// TwinCAT 3 PLC project NUCOIL
// libraries:
//   TcSUPS_CX51x0,newest,Evolution
//   YaskawaFunctions,newest,Evolution
//   Tc2_Drive, * (Beckhoff Automation GmbH)
//   Tc2_EtherCAT, * (Beckhoff Automation GmbH)
//   Tc2_IoFunctions, * (Beckhoff Automation GmbH)
//   Tc2_Math, * (Beckhoff Automation GmbH)
//   Tc2_MC2, * (Beckhoff Automation GmbH)
//   Tc2_MC2_Camming, * (Beckhoff Automation GmbH)
//   Tc2_NC, * (Beckhoff Automation GmbH)
//   Tc2_Standard, * (Beckhoff Automation GmbH)
//   Tc2_System, * (Beckhoff Automation GmbH)
//   Tc2_Utilities, * (Beckhoff Automation GmbH)
//   Tc3_Module, * (Beckhoff Automation GmbH)
// project tree:
//   Data types/ ST_AirTableBuf.TcDUT, ST_AlertLight.TcDUT, ST_AnaInput.TcDUT, ST_AxisPosBuf.TcDUT, ST_AxisTableBuf.TcDUT, ST_AxisTrqBuf.TcDUT, ST_AxisVelBuf.TcDUT, ST_BrakeParam.TcDUT, ST_Cam.TcDUT, ST_CamTable.TcDUT, ST_DigitInput.TcDUT, ST_DigitOutput.TcDUT, ST_DriveAlarmCode.TcDUT, ST_ExFSpdUpTableBuf.TcDUT, ST_FeederInProduce.TcDUT, ST_G5Config.TcDUT, ST_G5Status.TcDUT, ST_Homing.TcDUT, ST_InputState.TcDUT, ST_IOSwitch.TcDUT, ST_ManMove.TcDUT, ST_MasterAxisPos.TcDUT, ST_MasterAxisValue.TcDUT, ST_McFBInOutVar.TcDUT, ST_MCRelativeInput.TcDUT, ST_MCRelativeOutput.TcDUT, ST_McValue.TcDUT, ST_OIL.TcDUT, ST_OneLineAir.TcDUT, ST_OneLineTable.TcDUT, ST_ProAndManRelativeState.TcDUT, ST_Produce.TcDUT, ST_RingBuffer.TcDUT, ST_RingBufferIO.TcDUT, ST_RingBufferIOPart.TcDUT, ST_RingBufferPart.TcDUT, ST_SetPosByUI.TcDUT, ST_SlaveEcData.TcDUT, ST_SubProgramConfig.TcDUT, ST_SubProgramTable.TcDUT, ST_Touch.TcDUT, ST_TouchAdjustConfig.TcDUT, ST_TouchConfig.TcDUT, ST_TouchProbe.TcDUT, ST_TouchProbeHomeByUI.TcDUT, ST_TouchTableBuf.TcDUT
//   Global Variables/ ENUMSTATE.TcDUT, Global_Variables.TcGVL, MachineSubTypeEnum.TcDUT, MachineTypeEnum.TcDUT, MANMOVEENUM.TcDUT, MotorVenderEnum.TcDUT, Variable_Configuration.TcGVL
//   POUs/ AlertLight.TcPOU, AxisStatusDataStore.TcPOU, CoEConfig.TcPOU, CommunicationQualityCheck.TcPOU, EMGStop.TcPOU, EncoderClear.TcPOU, Error.TcPOU, HomeByTouchProbe.TcPOU, IOMapping.TcPOU, MAIN.TcPOU, ManMove.TcPOU, MCRelativeMove.TcPOU, MoveToColPos.TcPOU, Mpg.TcPOU, prAxis.TcPOU, Produce.TcPOU, SetCountPosToActPos.TcPOU, SetOverride.TcPOU, SetPosByUI.TcPOU, SubRunAlone.TcPOU, UPS.TcPOU
//   POUs/FB/ AlarmListClear.TcPOU, FB_CheckInfoData.TcPOU, FB_CloseAir.TcPOU, FB_CloseIO.TcPOU, FB_CloseOil.TcPOU, FB_EcAbnormal.TcPOU, FB_EncoderClear.TcPOU, FB_FNeedHoldPos.TcPOU, FB_GetExtPosition.TcPOU, FB_GetMachineInfo.TcPOU, FB_InAnotherTouch.TcPOU, FB_IsAdjustAxis.TcPOU, FB_IsAdjustTouch.TcPOU, FB_PosNear.TcPOU, FB_ToubleShootIsError.TcPOU, FB_TouchEnd.TcPOU, FB_TouchProbe.TcPOU, ManMovCal.TcPOU, MasterMove.TcPOU, MasterMove2.TcPOU, PPMCal.TcPOU, RelativeMOVE.TcPOU, RelativeMOVE2.TcPOU, SetMotionFuction.TcPOU, SetPositionTable.TcPOU
//   / Standard.TcTTO
// real-time tasks:
//   TASK Standard: cycle T#1ms, priority 25, ADS port 350
// motion (NC):
//   TASK NC-Task 1 SAF: cycle T#1ms, priority 4, ADS port 501
//   TASK NC-Task 1 SVB: cycle T#10ms, priority 8, ADS port 511
//   AXIS Axis1 Slide1 (id 2)
//     Dynamic: AccelerationMaximum=0, DecelerationMaximum=0, Acceleration=233017000, Deceleration=233017000, Jerk=124275000000
//     Velo: Maximum=6553600
//     PositionAreaControl: Enable=false
//     TargetPosControl: Enable=false
//     encoder EncType=1
//       EncPara: ScaleFactorNumerator=1
//     drive DrvType=5
//       DrvPara: DriveControlDWord=#x00000001
//         Analog: VeloReferenz=6553600, TorqueSetpointScale=10, SmoothingFilterOrder=0, SmoothingFilterTime=0
//         TimeComp: TaskDelayCycles=1
//     controller CtrType=1
//       CtrPara: PriorControlFactor=1
//         PosDiffControl: Enable=false
//         Observer: BandWidth=20
//   AXIS Axis2 Slide2 (id 3)
//     Dynamic: AccelerationMaximum=0, DecelerationMaximum=0, Acceleration=699050750.00009, Deceleration=699050750.00009, Jerk=1118479200001.57
//     Velo: Maximum=6553600
//     PositionAreaControl: Enable=false
//     TargetPosControl: Enable=false
//     encoder EncType=1
//       EncPara: ScaleFactorNumerator=1
//     drive DrvType=5
//       DrvPara: DriveControlDWord=#x00000001
//         Analog: VeloReferenz=6553600, TorqueSetpointScale=10, SmoothingFilterOrder=0, SmoothingFilterTime=0
//         TimeComp: TaskDelayCycles=1
//     controller CtrType=1
//       CtrPara: PriorControlFactor=1
//         PosDiffControl: Enable=false
//         Observer: BandWidth=20
//   AXIS Axis3 Slide3 (id 4)
//     Dynamic: AccelerationMaximum=0, DecelerationMaximum=0, Acceleration=3019980000, Deceleration=3019980000, Jerk=3025310000000
//     Velo: Maximum=6553600
//     PositionAreaControl: Enable=false
//     TargetPosControl: Enable=false
//     encoder EncType=1
//       EncPara: ScaleFactorNumerator=1
//     drive DrvType=5
//       DrvPara: DriveControlDWord=#x00000001
//         Analog: VeloReferenz=6553600, TorqueSetpointScale=10, SmoothingFilterOrder=0, SmoothingFilterTime=0
//         TimeComp: TaskDelayCycles=1
//     controller CtrType=1
//       CtrPara: PriorControlFactor=1
//         PosDiffControl: Enable=false
//         Observer: BandWidth=20
//   AXIS Axis4 Slide4 (id 5)
//     Dynamic: AccelerationMaximum=0, DecelerationMaximum=0, Acceleration=2206380000, Deceleration=2206380000, Jerk=11142200000000
//     Velo: Maximum=6553600
//     PositionAreaControl: Enable=false
//     TargetPosControl: Enable=false
//     encoder EncType=1
//       EncPara: ScaleFactorNumerator=1
//     drive DrvType=5
//       DrvPara: DriveControlDWord=#x00000001
//         Analog: VeloReferenz=6553600, TorqueSetpointScale=10, SmoothingFilterOrder=0, SmoothingFilterTime=0
//         TimeComp: TaskDelayCycles=1
//     controller CtrType=1
//       CtrPara: PriorControlFactor=1
//         PosDiffControl: Enable=false
//         Observer: BandWidth=20
//   AXIS Axis5 Slide5 (id 6)
//     Dynamic: AccelerationMaximum=0, DecelerationMaximum=0, Acceleration=441276000, Deceleration=441276000, Jerk=2971260000000
//     Velo: Maximum=6553600
//     PositionAreaControl: Enable=false
//     TargetPosControl: Enable=false
//     encoder EncType=1
//       EncPara: ScaleFactorNumerator=1
//     drive DrvType=5
//       DrvPara: DriveControlDWord=#x00000001
//         Analog: VeloReferenz=6553600, TorqueSetpointScale=10, SmoothingFilterOrder=0, SmoothingFilterTime=0
//         TimeComp: TaskDelayCycles=1
//     controller CtrType=1
//       CtrPara: PriorControlFactor=1
//         PosDiffControl: Enable=false
//         Observer: BandWidth=20
//   AXIS Axis6 Slide6 (id 7)
//     Dynamic: AccelerationMaximum=0, DecelerationMaximum=0, Acceleration=2206380000, Deceleration=2206380000, Jerk=11142200000000
//     Velo: Maximum=6553600
//     PositionAreaControl: Enable=false
//     TargetPosControl: Enable=false
//     encoder EncType=1
//       EncPara: ScaleFactorNumerator=1
//     drive DrvType=5
//       DrvPara: DriveControlDWord=#x00000001
//         Analog: VeloReferenz=6553600, TorqueSetpointScale=10, SmoothingFilterOrder=0, SmoothingFilterTime=0
//         TimeComp: TaskDelayCycles=1
//     controller CtrType=1
//       CtrPara: PriorControlFactor=1
//         PosDiffControl: Enable=false
//         Observer: BandWidth=20
//   AXIS Axis7 Slide7 (id 8)
//     Dynamic: AccelerationMaximum=0, DecelerationMaximum=0, Acceleration=2206376778.77214, Deceleration=2206376778.77214, Jerk=11142167465677.8
//     Velo: Maximum=6553600
//     PositionAreaControl: Enable=false
//     TargetPosControl: Enable=false
//     encoder EncType=1
//       EncPara: ScaleFactorNumerator=1
//     drive DrvType=5
//       DrvPara: DriveControlDWord=#x00000001
//         Analog: VeloReferenz=6553600, TorqueSetpointScale=10, SmoothingFilterOrder=0, SmoothingFilterTime=0
//         TimeComp: TaskDelayCycles=1
//     controller CtrType=1
//       CtrPara: PriorControlFactor=1
//         PosDiffControl: Enable=false
//         Observer: BandWidth=20
//   AXIS Axis8 Slide8 (id 9)
//     Dynamic: AccelerationMaximum=0, DecelerationMaximum=0, Acceleration=2206376778.77214, Deceleration=2206376778.77214, Jerk=11142167465677.8
//     Velo: Maximum=6553600
//     PositionAreaControl: Enable=false
//     TargetPosControl: Enable=false
//     encoder EncType=1
//       EncPara: ScaleFactorNumerator=1
//     drive DrvType=5
//       DrvPara: DriveControlDWord=#x00000001
//         Analog: VeloReferenz=6553600, TorqueSetpointScale=10, SmoothingFilterOrder=0, SmoothingFilterTime=0
//         TimeComp: TaskDelayCycles=1
//     controller CtrType=1
//       CtrPara: PriorControlFactor=1
//         PosDiffControl: Enable=false
//         Observer: BandWidth=20
//   AXIS Axis9 Wire (id 10)
//     Dynamic: AccelerationMaximum=0, DecelerationMaximum=0, Acceleration=2206376778.77214, Deceleration=2206376778.77214, Jerk=11142167465677.8
//     Velo: Maximum=6553600
//     PositionAreaControl: Enable=false
//     TargetPosControl: Enable=false
//     encoder EncType=1
//       EncPara: ScaleFactorNumerator=1
//     drive DrvType=5
//       DrvPara: DriveControlDWord=#x00000001
//         Analog: VeloReferenz=6553600, TorqueSetpointScale=10, SmoothingFilterOrder=0, SmoothingFilterTime=0
//         TimeComp: TaskDelayCycles=1
//     controller CtrType=1
//       CtrPara: PriorControlFactor=1
//         PosDiffControl: Enable=false
//         Observer: BandWidth=20
//   AXIS Axis10 RWire (id 11)
//     Dynamic: AccelerationMaximum=0, DecelerationMaximum=0, Acceleration=2206376778.77214, Deceleration=2206376778.77214, Jerk=11142167465677.8
//     Velo: Maximum=6553600
//     PositionAreaControl: Enable=false
//     TargetPosControl: Enable=false
//     encoder EncType=1
//       EncPara: ScaleFactorNumerator=1
//     drive DrvType=5
//       DrvPara: DriveControlDWord=#x00000001
//         Analog: VeloReferenz=6553600, TorqueSetpointScale=10, SmoothingFilterOrder=0, SmoothingFilterTime=0
//         TimeComp: TaskDelayCycles=1
//     controller CtrType=1
//       CtrPara: PriorControlFactor=1
//         PosDiffControl: Enable=false
//         Observer: BandWidth=20
//   AXIS Axis11 Quil (id 12)
//     Dynamic: AccelerationMaximum=0, DecelerationMaximum=0, Acceleration=2206376778.77214, Deceleration=2206376778.77214, Jerk=11142167465677.8
//     Velo: Maximum=6553600
//     PositionAreaControl: Enable=false
//     TargetPosControl: Enable=false
//     encoder EncType=1
//       EncPara: ScaleFactorNumerator=1
//     drive DrvType=5
//       DrvPara: DriveControlDWord=#x00000001
//         Analog: VeloReferenz=6553600, TorqueSetpointScale=10, SmoothingFilterOrder=0, SmoothingFilterTime=0
//         TimeComp: TaskDelayCycles=1
//     controller CtrType=1
//       CtrPara: PriorControlFactor=1
//         PosDiffControl: Enable=false
//         Observer: BandWidth=20
//   AXIS Axis12 X (id 13)
//     Dynamic: AccelerationMaximum=0, DecelerationMaximum=0, Acceleration=2206380000, Deceleration=2206380000, Jerk=11142200000000
//     Velo: Maximum=6553600
//     PositionAreaControl: Enable=false
//     TargetPosControl: Enable=false
//     encoder EncType=1
//       EncPara: ScaleFactorNumerator=1
//     drive DrvType=5
//       DrvPara: DriveControlDWord=#x00000001
//         Analog: VeloReferenz=6553600, TorqueSetpointScale=10, SmoothingFilterOrder=0, SmoothingFilterTime=0
//         TimeComp: TaskDelayCycles=1
//     controller CtrType=1
//       CtrPara: PriorControlFactor=1
//         PosDiffControl: Enable=false
//         Observer: BandWidth=20
//   AXIS Axis13 Y (id 14)
//     Dynamic: AccelerationMaximum=0, DecelerationMaximum=0, Acceleration=2206380000, Deceleration=2206380000, Jerk=11142200000000
//     Velo: Maximum=6553600
//     PositionAreaControl: Enable=false
//     TargetPosControl: Enable=false
//     encoder EncType=1
//       EncPara: ScaleFactorNumerator=1
//     drive DrvType=5
//       DrvPara: DriveControlDWord=#x00000001
//         Analog: VeloReferenz=6553600, TorqueSetpointScale=10, SmoothingFilterOrder=0, SmoothingFilterTime=0
//         TimeComp: TaskDelayCycles=1
//     controller CtrType=1
//       CtrPara: PriorControlFactor=1
//         PosDiffControl: Enable=false
//         Observer: BandWidth=20
//   AXIS Axis14 Z (id 15)
//     Dynamic: AccelerationMaximum=0, DecelerationMaximum=0, Acceleration=2206380000, Deceleration=2206380000, Jerk=11142200000000
//     Velo: Maximum=6553600
//     PositionAreaControl: Enable=false
//     TargetPosControl: Enable=false
//     encoder EncType=1
//       EncPara: ScaleFactorNumerator=1
//     drive DrvType=5
//       DrvPara: DriveControlDWord=#x00000001
//         Analog: VeloReferenz=6553600, TorqueSetpointScale=10, SmoothingFilterOrder=0, SmoothingFilterTime=0
//         TimeComp: TaskDelayCycles=1
//     controller CtrType=1
//       CtrPara: PriorControlFactor=1
//         PosDiffControl: Enable=false
//         Observer: BandWidth=20
//   AXIS Axis15 Rtool (id 16)
//     Dynamic: AccelerationMaximum=0, DecelerationMaximum=0, Acceleration=2206380000, Deceleration=2206380000, Jerk=11142200000000
//     Velo: Maximum=6553600
//     PositionAreaControl: Enable=false
//     TargetPosControl: Enable=false
//     encoder EncType=1
//       EncPara: ScaleFactorNumerator=1
//     drive DrvType=5
//       DrvPara: DriveControlDWord=#x00000001
//         Analog: VeloReferenz=6553600, TorqueSetpointScale=10, SmoothingFilterOrder=0, SmoothingFilterTime=0
//         TimeComp: TaskDelayCycles=1
//     controller CtrType=1
//       CtrPara: PriorControlFactor=1
//         PosDiffControl: Enable=false
//         Observer: BandWidth=20
//   AXIS Axis16 SpinA (id 17)
//     Dynamic: AccelerationMaximum=0, DecelerationMaximum=0, Acceleration=2206380000, Deceleration=2206380000, Jerk=11142200000000
//     Velo: Maximum=6553600
//     PositionAreaControl: Enable=false
//     TargetPosControl: Enable=false
//     encoder EncType=1
//       EncPara: ScaleFactorNumerator=1
//     drive DrvType=5
//       DrvPara: DriveControlDWord=#x00000001
//         Analog: VeloReferenz=6553600, TorqueSetpointScale=10, SmoothingFilterOrder=0, SmoothingFilterTime=0
//         TimeComp: TaskDelayCycles=1
//     controller CtrType=1
//       CtrPara: PriorControlFactor=1
//         PosDiffControl: Enable=false
//         Observer: BandWidth=20
//   AXIS Axis17 SpinB (id 18)
//     Dynamic: AccelerationMaximum=0, DecelerationMaximum=0, Acceleration=2206380000, Deceleration=2206380000, Jerk=11142200000000
//     Velo: Maximum=6553600
//     PositionAreaControl: Enable=false
//     TargetPosControl: Enable=false
//     encoder EncType=1
//       EncPara: ScaleFactorNumerator=1
//     drive DrvType=5
//       DrvPara: DriveControlDWord=#x00000001
//         Analog: VeloReferenz=6553600, TorqueSetpointScale=10, SmoothingFilterOrder=0, SmoothingFilterTime=0
//         TimeComp: TaskDelayCycles=1
//     controller CtrType=1
//       CtrPara: PriorControlFactor=1
//         PosDiffControl: Enable=false
//         Observer: BandWidth=20
//   AXIS Axis18 SpinC (id 19)
//     Dynamic: AccelerationMaximum=0, DecelerationMaximum=0, Acceleration=2206380000, Deceleration=2206380000, Jerk=11142200000000
//     Velo: Maximum=6553600
//     PositionAreaControl: Enable=false
//     TargetPosControl: Enable=false
//     encoder EncType=1
//       EncPara: ScaleFactorNumerator=1
//     drive DrvType=5
//       DrvPara: DriveControlDWord=#x00000001
//         Analog: VeloReferenz=6553600, TorqueSetpointScale=10, SmoothingFilterOrder=0, SmoothingFilterTime=0
//         TimeComp: TaskDelayCycles=1
//     controller CtrType=1
//       CtrPara: PriorControlFactor=1
//         PosDiffControl: Enable=false
//         Observer: BandWidth=20
//   AXIS Axis19 SpinD (id 20)
//     Dynamic: AccelerationMaximum=0, DecelerationMaximum=0, Acceleration=2206380000, Deceleration=2206380000, Jerk=11142200000000
//     Velo: Maximum=6553600
//     PositionAreaControl: Enable=false
//     TargetPosControl: Enable=false
//     encoder EncType=1
//       EncPara: ScaleFactorNumerator=1
//     drive DrvType=5
//       DrvPara: DriveControlDWord=#x00000001
//         Analog: VeloReferenz=6553600, TorqueSetpointScale=10, SmoothingFilterOrder=0, SmoothingFilterTime=0
//         TimeComp: TaskDelayCycles=1
//     controller CtrType=1
//       CtrPara: PriorControlFactor=1
//         PosDiffControl: Enable=false
//         Observer: BandWidth=20
//   AXIS Axis20 SpinE (id 21)
//     Dynamic: AccelerationMaximum=0, DecelerationMaximum=0, Acceleration=2206380000, Deceleration=2206380000, Jerk=11142200000000
//     Velo: Maximum=6553600
//     PositionAreaControl: Enable=false
//     TargetPosControl: Enable=false
//     encoder EncType=1
//       EncPara: ScaleFactorNumerator=1
//     drive DrvType=5
//       DrvPara: DriveControlDWord=#x00000001
//         Analog: VeloReferenz=6553600, TorqueSetpointScale=10, SmoothingFilterOrder=0, SmoothingFilterTime=0
//         TimeComp: TaskDelayCycles=1
//     controller CtrType=1
//       CtrPara: PriorControlFactor=1
//         PosDiffControl: Enable=false
//         Observer: BandWidth=20
// I/O:
//   DEVICE Device 1 (EtherCAT) (disabled), AmsNetId 0.0.0.0.1.2
//     Term 1 (EK1100) [EK1100 EtherCAT Coupler (2A E-Bus)]
//       Term 2 (EL1889) [EL1889 16Ch. Dig. Input 24V, 3ms, negative]
//       Term 3 (EL1889) [EL1889 16Ch. Dig. Input 24V, 3ms, negative]
//       Term 4 (EL1889) [EL1889 16Ch. Dig. Input 24V, 3ms, negative]
//       Term 5 (EL1889) [EL1889 16Ch. Dig. Input 24V, 3ms, negative]
//       Term 6 (EL2889) [EL2889 16Ch. Dig. Output 24V, 0.5A, negative]
//       Term 7 (EL2889) [EL2889 16Ch. Dig. Output 24V, 0.5A, negative]
//       Term 8 (EL2889) [EL2889 16Ch. Dig. Output 24V, 0.5A, negative]
//       Term 9 (EL3062-0030) [EL3062-0030 2Ch. Ana. Input 0-30V]
//       Term 10 (EL5101) [EL5101 1Ch. Inc. Encoder 5V]
//       Term 11 (EK1110) [EK1110 EtherCAT extension]
//     Drive1 Slide1 (SanyoDenki RS2 EtherCAT) [R ADVANCED MODEL with EtherCAT(P0002813E01)]
//     Drive2 Slide2 (SanyoDenki RS2 EtherCAT) [R ADVANCED MODEL with EtherCAT(P0002813E01)]
//     Drive3 Slide3 (SanyoDenki RS2 EtherCAT) [R ADVANCED MODEL with EtherCAT(P0002813E01)]
//     Drive4 Slide4  (SanyoDenki RS2 EtherCAT) [R ADVANCED MODEL with EtherCAT(P0002813E01)]
//     Drive5 Slide5 (SanyoDenki RS2 EtherCAT) [R ADVANCED MODEL with EtherCAT(P0002813E01)]
//     Drive6 Slide6 (SanyoDenki RS2 EtherCAT) [R ADVANCED MODEL with EtherCAT(P0002813E01)]
//     Drive7 Slide7 (SanyoDenki RS2 EtherCAT) [R ADVANCED MODEL with EtherCAT(P0002813E01)]
//     Drive8 Slide8 (SanyoDenki RS2 EtherCAT) [R ADVANCED MODEL with EtherCAT(P0002813E01)]
//     Drive9 Wire (SanyoDenki RS2 EtherCAT) [R ADVANCED MODEL with EtherCAT(P0002813E01)]
//     Drive10 RWire (SanyoDenki RS2 EtherCAT) [R ADVANCED MODEL with EtherCAT(P0002813E01)]
//     Drive11 Quill  (SanyoDenki RS2 EtherCAT) [R ADVANCED MODEL with EtherCAT(P0002813E01)]
//     Drive12 X (SanyoDenki RS2 EtherCAT) [R ADVANCED MODEL with EtherCAT(P0002813E01)]
//     Drive13 Y (SanyoDenki RS2 EtherCAT) [R ADVANCED MODEL with EtherCAT(P0002813E01)]
//     Drive14 Z (SanyoDenki RS2 EtherCAT) [R ADVANCED MODEL with EtherCAT(P0002813E01)]
//     Drive15 Rtool (SanyoDenki RS2 EtherCAT) [R ADVANCED MODEL with EtherCAT(P0002813E01)]
//     Drive16 SpinA (SanyoDenki RS2 EtherCAT) [R ADVANCED MODEL with EtherCAT(P0002813E01)]
//     Drive17 SpinB (SanyoDenki RS2 EtherCAT) [R ADVANCED MODEL with EtherCAT(P0002813E01)]
//     Drive18 SpinC (SanyoDenki RS2 EtherCAT) [R ADVANCED MODEL with EtherCAT(P0002813E01)]
//     Drive19 SpinD (SanyoDenki RS2 EtherCAT) [R ADVANCED MODEL with EtherCAT(P0002813E01)]
//     Drive20 SpinE (SanyoDenki RS2 EtherCAT) [R ADVANCED MODEL with EtherCAT(P0002813E01)]
//     Drive21 DSpinA1 (SanyoDenki RS2 EtherCAT) [R ADVANCED MODEL with EtherCAT(P0002813E01)]
//     Drive22 DSpinA2 (SanyoDenki RS2 EtherCAT) [R ADVANCED MODEL with EtherCAT(P0002813E01)]
//     Drive23 DSpinB1 (SanyoDenki RS2 EtherCAT) [R ADVANCED MODEL with EtherCAT(P0002813E01)]
//     Drive24 DSpinB2 (SanyoDenki RS2 EtherCAT) [R ADVANCED MODEL with EtherCAT(P0002813E01)]
//     Drive25 DSpinC1 (SanyoDenki RS2 EtherCAT) [R ADVANCED MODEL with EtherCAT(P0002813E01)]
//     Drive26 DSpinC2 (SanyoDenki RS2 EtherCAT) [R ADVANCED MODEL with EtherCAT(P0002813E01)]
//     Drive27 DSpinD1 (SanyoDenki RS2 EtherCAT) [R ADVANCED MODEL with EtherCAT(P0002813E01)]
//     Drive28 DSpinD2 (SanyoDenki RS2 EtherCAT) [R ADVANCED MODEL with EtherCAT(P0002813E01)]
//     Drive29 SpinF (SanyoDenki RS2 EtherCAT) [R ADVANCED MODEL with EtherCAT(P0002813E01)]
//     Drive30 Cut (SanyoDenki RS2 EtherCAT) [R ADVANCED MODEL with EtherCAT(P0002813E01)]
// variable links:
//   NUCOIL/NUCOIL Instance <-> NC-Task 1 SAF/Axes/Axis1 Slide1
//     Standard Inputs/.Axis[1].Axis.NcToPlc <-> Outputs/Axis1 Slide1_ToPlc
//     Standard Outputs/.Axis[1].Axis.PlcToNc <-> Inputs/Axis1 Slide1_FromPlc
//   NUCOIL/NUCOIL Instance <-> NC-Task 1 SAF/Axes/Axis10 RWire
//     Standard Inputs/.Axis[10].Axis.NcToPlc <-> Outputs/Axis10 RWire_ToPlc
//     Standard Outputs/.Axis[10].Axis.PlcToNc <-> Inputs/Axis10 RWire_FromPlc
//   NUCOIL/NUCOIL Instance <-> NC-Task 1 SAF/Axes/Axis11 Quil
//     Standard Inputs/.Axis[11].Axis.NcToPlc <-> Outputs/Axis11 Quil_ToPlc
//     Standard Outputs/.Axis[11].Axis.PlcToNc <-> Inputs/Axis11 Quil_FromPlc
//   NUCOIL/NUCOIL Instance <-> NC-Task 1 SAF/Axes/Axis12 X
//     Standard Inputs/.Axis[12].Axis.NcToPlc <-> Outputs/Axis12 X_ToPlc
//     Standard Outputs/.Axis[12].Axis.PlcToNc <-> Inputs/Axis12 X_FromPlc
//   NUCOIL/NUCOIL Instance <-> NC-Task 1 SAF/Axes/Axis13 Y
//     Standard Inputs/.Axis[13].Axis.NcToPlc <-> Outputs/Axis13 Y_ToPlc
//     Standard Outputs/.Axis[13].Axis.PlcToNc <-> Inputs/Axis13 Y_FromPlc
//   NUCOIL/NUCOIL Instance <-> NC-Task 1 SAF/Axes/Axis14 Z
//     Standard Inputs/.Axis[14].Axis.NcToPlc <-> Outputs/Axis14 Z_ToPlc
//     Standard Outputs/.Axis[14].Axis.PlcToNc <-> Inputs/Axis14 Z_FromPlc
//   NUCOIL/NUCOIL Instance <-> NC-Task 1 SAF/Axes/Axis15 Rtool
//     Standard Inputs/.Axis[15].Axis.NcToPlc <-> Outputs/Axis15 Rtool_ToPlc
//     Standard Outputs/.Axis[15].Axis.PlcToNc <-> Inputs/Axis15 Rtool_FromPlc
//   NUCOIL/NUCOIL Instance <-> NC-Task 1 SAF/Axes/Axis16 SpinA
//     Standard Inputs/.Axis[16].Axis.NcToPlc <-> Outputs/Axis16 SpinA_ToPlc
//     Standard Outputs/.Axis[16].Axis.PlcToNc <-> Inputs/Axis16 SpinA_FromPlc
//   NUCOIL/NUCOIL Instance <-> NC-Task 1 SAF/Axes/Axis17 SpinB
//     Standard Inputs/.Axis[17].Axis.NcToPlc <-> Outputs/Axis17 SpinB_ToPlc
//     Standard Outputs/.Axis[17].Axis.PlcToNc <-> Inputs/Axis17 SpinB_FromPlc
//   NUCOIL/NUCOIL Instance <-> NC-Task 1 SAF/Axes/Axis18 SpinC
//     Standard Inputs/.Axis[18].Axis.NcToPlc <-> Outputs/Axis18 SpinC_ToPlc
//     Standard Outputs/.Axis[18].Axis.PlcToNc <-> Inputs/Axis18 SpinC_FromPlc
//   NUCOIL/NUCOIL Instance <-> NC-Task 1 SAF/Axes/Axis19 SpinD
//     Standard Inputs/.Axis[19].Axis.NcToPlc <-> Outputs/Axis19 SpinD_ToPlc
//     Standard Outputs/.Axis[19].Axis.PlcToNc <-> Inputs/Axis19 SpinD_FromPlc
//   NUCOIL/NUCOIL Instance <-> NC-Task 1 SAF/Axes/Axis2 Slide2
//     Standard Inputs/.Axis[2].Axis.NcToPlc <-> Outputs/Axis2 Slide2_ToPlc
//     Standard Outputs/.Axis[2].Axis.PlcToNc <-> Inputs/Axis2 Slide2_FromPlc
//   NUCOIL/NUCOIL Instance <-> NC-Task 1 SAF/Axes/Axis20 SpinE
//     Standard Inputs/.Axis[20].Axis.NcToPlc <-> Outputs/Axis20 SpinE_ToPlc
//     Standard Outputs/.Axis[20].Axis.PlcToNc <-> Inputs/Axis20 SpinE_FromPlc
//   NUCOIL/NUCOIL Instance <-> NC-Task 1 SAF/Axes/Axis3 Slide3
//     Standard Inputs/.Axis[3].Axis.NcToPlc <-> Outputs/Axis3 Slide3_ToPlc
//     Standard Outputs/.Axis[3].Axis.PlcToNc <-> Inputs/Axis3 Slide3_FromPlc
//   NUCOIL/NUCOIL Instance <-> NC-Task 1 SAF/Axes/Axis4 Slide4
//     Standard Inputs/.Axis[4].Axis.NcToPlc <-> Outputs/Axis4 Slide4_ToPlc
//     Standard Outputs/.Axis[4].Axis.PlcToNc <-> Inputs/Axis4 Slide4_FromPlc
//   NUCOIL/NUCOIL Instance <-> NC-Task 1 SAF/Axes/Axis5 Slide5
//     Standard Inputs/.Axis[5].Axis.NcToPlc <-> Outputs/Axis5 Slide5_ToPlc
//     Standard Outputs/.Axis[5].Axis.PlcToNc <-> Inputs/Axis5 Slide5_FromPlc
//   NUCOIL/NUCOIL Instance <-> NC-Task 1 SAF/Axes/Axis6 Slide6
//     Standard Inputs/.Axis[6].Axis.NcToPlc <-> Outputs/Axis6 Slide6_ToPlc
//     Standard Outputs/.Axis[6].Axis.PlcToNc <-> Inputs/Axis6 Slide6_FromPlc
//   NUCOIL/NUCOIL Instance <-> NC-Task 1 SAF/Axes/Axis7 Slide7
//     Standard Inputs/.Axis[7].Axis.NcToPlc <-> Outputs/Axis7 Slide7_ToPlc
//     Standard Outputs/.Axis[7].Axis.PlcToNc <-> Inputs/Axis7 Slide7_FromPlc
//   NUCOIL/NUCOIL Instance <-> NC-Task 1 SAF/Axes/Axis8 Slide8
//     Standard Inputs/.Axis[8].Axis.NcToPlc <-> Outputs/Axis8 Slide8_ToPlc
//     Standard Outputs/.Axis[8].Axis.PlcToNc <-> Inputs/Axis8 Slide8_FromPlc
//   NUCOIL/NUCOIL Instance <-> NC-Task 1 SAF/Axes/Axis9 Wire
//     Standard Inputs/.Axis[9].Axis.NcToPlc <-> Outputs/Axis9 Wire_ToPlc
//     Standard Outputs/.Axis[9].Axis.PlcToNc <-> Inputs/Axis9 Wire_FromPlc

CONFIGURATION NUCOIL
    RESOURCE PLC ON TwinCAT3
        TASK Standard(INTERVAL := T#1ms, PRIORITY := 25);
        PROGRAM MAIN WITH Standard : MAIN;
    END_RESOURCE
END_CONFIGURATION

// ---- Data types/ST_AirTableBuf.TcDUT
TYPE ST_AirTableBuf :
STRUCT
	Table	: ARRAY [1..AirNo, 0..1999] OF BOOL;
	OK		: BOOL;
END_STRUCT
END_TYPE

// ---- Data types/ST_AlertLight.TcDUT
TYPE ST_AlertLight :
STRUCT
	Orange  : BOOL;
    Green   : BOOL;
    Red     : BOOL;
END_STRUCT
END_TYPE

// ---- Data types/ST_AnaInput.TcDUT
TYPE ST_AnaInput :
STRUCT
	Input	: ARRAY[0..3] OF INT;
END_STRUCT
END_TYPE

// ---- Data types/ST_AxisPosBuf.TcDUT
TYPE ST_AxisPosBuf :
STRUCT
	SetPos	: ARRAY [0..999] OF LREAL;
    ActPos  : ARRAY [0..999] OF LREAL;
END_STRUCT
END_TYPE

// ---- Data types/ST_AxisTableBuf.TcDUT
{attribute 'pack_mode' := '1'} 
TYPE ST_AxisTableBuf :
STRUCT
	Table	: ARRAY [1..No, 0..1999] OF LREAL;
	OK		: BOOL;
END_STRUCT
END_TYPE

// ---- Data types/ST_AxisTrqBuf.TcDUT
TYPE ST_AxisTrqBuf :
STRUCT
	Trq  : ARRAY [0..999] OF INT;
END_STRUCT
END_TYPE

// ---- Data types/ST_AxisVelBuf.TcDUT
TYPE ST_AxisVelBuf :
STRUCT
	SetVel  : ARRAY [0..999] OF LREAL;
	ActVel  : ARRAY [0..999] OF LREAL;
END_STRUCT
END_TYPE

// ---- Data types/ST_BrakeParam.TcDUT
TYPE ST_BrakeParam :
STRUCT
	Deceleration 	: LREAL;
	Jerk 		: LREAL;
END_STRUCT
END_TYPE

// ---- Data types/ST_Cam.TcDUT
TYPE ST_Cam :
STRUCT
	CamIn			: MC_CamIn_V2;
	CamOut			: MC_CamOut;
	TableSelect   		: MC_CamTableSelect;
	TableSelect2		: MC_CamTableSelect;
	Table	         		: MC_CAM_REF;
	Table2	         		: MC_CAM_REF;
	MotionFunction 	: ARRAY[1..10] OF MC_MotionFunctionPoint;
	Scaling 			: ST_CamScalingData;
	Options			:ST_CamInOptions_V2;
END_STRUCT
END_TYPE

// ---- Data types/ST_CamTable.TcDUT
TYPE ST_CamTable :
STRUCT
	PositionTable		: ARRAY[1..3600, 1..2] OF LREAL;
	NoOfRows			: UDINT;
	boolbuf1				: BOOL;
	boolbuf2				: BOOL;
	boolbuf3				: BOOL;
	boolbuf4				: BOOL;
END_STRUCT
END_TYPE

// ---- Data types/ST_DigitInput.TcDUT
TYPE ST_DigitInput :
STRUCT
	Input		: ARRAY[1..16] OF BOOL;
END_STRUCT
END_TYPE

// ---- Data types/ST_DigitOutput.TcDUT
TYPE ST_DigitOutput :
STRUCT
	Output 	: ARRAY[1..16] OF BOOL;
END_STRUCT
END_TYPE

// ---- Data types/ST_DriveAlarmCode.TcDUT
TYPE ST_DriveAlarmCode :
STRUCT
	Error1	: USINT;
	Error2	: USINT;
	Error3	: USINT;
	Error4	: USINT;
END_STRUCT
END_TYPE

// ---- Data types/ST_ExFSpdUpTableBuf.TcDUT
TYPE ST_ExFSpdUpTableBuf :
STRUCT
	Table	: ARRAY [0..1999] OF BOOL;
	OK		: BOOL;
END_STRUCT
END_TYPE

// ---- Data types/ST_FeederInProduce.TcDUT
TYPE ST_FeederInProduce :
STRUCT
	CurPos			: LREAL;
	BasePos 		: LREAL;

	StillPos			: LREAL;
	TouchPos		: LREAL;
	TouchFeederIdx	: INT;

END_STRUCT
END_TYPE

// ---- Data types/ST_G5Config.TcDUT
TYPE ST_G5Config :
STRUCT
	ATime		: UDINT;
	BTime		: UDINT;
	RepeatTimes :UINT;
END_STRUCT
END_TYPE

// ---- Data types/ST_G5Status.TcDUT
TYPE ST_G5Status :
STRUCT
	CurIdx				:INT;
	CurTimes			:INT;
	ATimeFIdx			:INT;
	ATimeSubNo			:INT;
	JumpFirstTime 		:BOOL;
	ATimeTouchConfigIdx	: ARRAY [1..TouchNo] OF INT;
END_STRUCT
END_TYPE

// ---- Data types/ST_Homing.TcDUT
TYPE ST_Homing :
STRUCT
	Mode		: SINT;
	FirstSpd		: UDINT;
	SecSpd		: UDINT;
	AccSpd		: UDINT;
END_STRUCT
END_TYPE

// ---- Data types/ST_InputState.TcDUT
TYPE ST_InputState :
STRUCT
(*-------------------------------------Input1--------------------------------------*)
	PowerOff		:BOOL;
	Reset		    :BOOL;
	Producing		:BOOL;
	Testing			:BOOL;
	EditLock		:BOOL;
	ExFeederError	:BOOL;
	SafetyError		:BOOL;
	OilError		:BOOL;
	VRSwitch		:BOOL;
	EMGStop			:BOOL;
	HomeA			:BOOL;
	plusA			:BOOL;
	negA			:BOOL;
	plusY			:BOOL;
	negY			:BOOL;
	SW				:BOOL;

(*-------------------------------------Input2--------------------------------------*)
	Touch1			:BOOL;
	Touch2			:BOOL;
	Touch3			:BOOL;
	Touch4			:BOOL;
	StopCycle		:BOOL;
	ExDeviceError	:BOOL;
	PowerBit0		:BOOL;
	PowerBit1		:BOOL;
	ChoiceAxisBit0	:BOOL;
	ChoiceAxisBit1	:BOOL;
	ChoiceAxisBit2	:BOOL;
	ChoiceAxisBit3	:BOOL;
	ChoiceAxisBit4	:BOOL;
	FAlarm_1370		:BOOL;
	
(*-------------------------------------Input3--------------------------------------*)
	NG				:BOOL;
	Mpg_PositiveBtn	:BOOL;
	Mpg_NegativeBtn	:BOOL;
	Zrt				:BOOL;

(*-------------------------------------Input4--------------------------------------*)
	SafetyError1	:BOOL;
	SafetyError2	:BOOL;
	SafetyError3	:BOOL;
	SafetyError4	:BOOL;
	PanelEStop		:BOOL;
	FrontEStop		:BOOL;
	SideEStop		:BOOL;
	RearEStop		:BOOL;
	DecoilorEStop   :BOOL;

END_STRUCT
END_TYPE

// ---- Data types/ST_IOSwitch.TcDUT
TYPE ST_IOSwitch :
STRUCT
	SaftyEnable			:BOOL;
	SafetyLockDisable   :BOOL;
	GlobalTouchEnable   :BOOL;
END_STRUCT
END_TYPE

// ---- Data types/ST_ManMove.TcDUT
TYPE ST_ManMove :
STRUCT
	 DistByUnit		:LREAL;
	 UnitRatio		:LREAL;
	 JerkP			:LREAL;
	 MoveTime 		:LREAL;
	 AccTime		:LREAL;
	Execute			:BOOL;
	boolbuf1			:BOOL;
	boolbuf2			:BOOL;
	boolbuf3			:BOOL;
	boolbuf4			:BOOL;
	boolbuf5			:BOOL;
	boolbuf6			:BOOL;
	boolbuf7			:BOOL;
END_STRUCT
END_TYPE

// ---- Data types/ST_MasterAxisPos.TcDUT
TYPE ST_MasterAxisPos :
STRUCT
	Pos		: DINT:=0;
	PosLast 	: DINT:=0;
END_STRUCT
END_TYPE

// ---- Data types/ST_MasterAxisValue.TcDUT
TYPE ST_MasterAxisValue :
STRUCT
	Distance			: LREAL;
	Velocity			: LREAL;
	TPhase1			: LREAL;
	TPhase2			: LREAL;
	Acceleration		: LREAL;
	Deceleration		: LREAL;
	Jerk				: LREAL;
	Idx				: INT:=1;
END_STRUCT
END_TYPE

// ---- Data types/ST_McFBInOutVar.TcDUT
TYPE ST_McFBInOutVar :
STRUCT
	Axis					:AXIS_REF;
	ActPos					: LREAL;

	fb_MC_ReadActualPosition :MC_ReadActualPosition;
	fbMC_Power				:MC_Power;
	fbMC_MoveRelative		:ARRAY [1..2] OF MC_MoveRelative;
	fbMC_ReadStatus			:MC_ReadStatus;
	fbMC_SetPosition		:MC_SetPosition;
	fbMC_Jog				:MC_Jog;
	fbMC_TouchProbe			:MC_TouchProbe;
	fbMC_Reset				:MC_Reset;
	fbMC_SetOverride		:MC_SetOverride;

	EnableSetPointGenerator	:MC_ExtSetPointGenEnable;
	DisableSetPointGenerator:MC_ExtSetPointGenDisable;

	fbSDOWrite 				:FB_EcCoESdoWriteEx;
	fbSDOWrite2 			:FB_EcCoESdoWriteEx;
	fbSDORead				:FB_EcCoESdoReadEx;
	fbADSWrite				:ADSWRITE;

	stPowerMcOutputs		: ST_McOutputs;
	stRelativeMcOutputs		: ARRAY [1..2] OF ST_McOutputs;
END_STRUCT
END_TYPE

// ---- Data types/ST_MCRelativeInput.TcDUT
TYPE ST_MCRelativeInput :
STRUCT
	Distance			:LREAL;
	Velocity  			:LREAL;
	Acceleration  		:LREAL;
	Deceleration 	 	:LREAL;
	Jerk				:LREAL;
	Execute  			:BOOL:=FALSE;
	boolbuf1			:BOOL;
	boolbuf2			:BOOL;
	boolbuf3			:BOOL;
	boolbuf4			:BOOL;
	boolbuf5			:BOOL;
	boolbuf6			:BOOL;
	boolbuf7			:BOOL;
END_STRUCT
END_TYPE

// ---- Data types/ST_MCRelativeOutput.TcDUT
TYPE ST_MCRelativeOutput :
STRUCT
	Done 				:BOOL;
	Busy 				:BOOL;
	Active 				:BOOL;
	CommandAborted 	:BOOL;
	Error 				:BOOL;
	boolbuf1				:BOOL;
	boolbuf2				:BOOL;
	boolbuf3				:BOOL;
	ErrorID 				:UDINT;
END_STRUCT
END_TYPE

// ---- Data types/ST_McValue.TcDUT
TYPE ST_McValue :
STRUCT
	Pos_360				: LREAL := 0;

	MoveExecute			:ARRAY [1..2] OF BOOL;
	MoveDistance		:ARRAY [1..2] OF LREAL;
	MoveVelocity			:ARRAY [1..2] OF LREAL;
	MoveAcceleration		:ARRAY [1..2] OF LREAL;
	MoveDeceleration		:ARRAY [1..2] OF LREAL;
	MoveJerk			:ARRAY [1..2] OF LREAL;

	Jog_JogForward		:BOOL;
	Jog_JogBackwards	:BOOL;
	Jog_Mode			:E_JogMode;
	Jog_Position			:LREAL;
	Jog_Velocity			:LREAL;
	Jog_Acceleration		:LREAL;
	Jog_Deceleration		:LREAL;
	Jog_Jerk			:LREAL;

END_STRUCT
END_TYPE

// ---- Data types/ST_OIL.TcDUT
TYPE ST_OIL :
STRUCT
	OpenTime	: UDINT;
	CloseTime	: UDINT;
	CurTime		: UDINT;
	CloseStrokes : UDINT;
	CurStrokes 	: UDINT;
	IsOpen		: BOOL:=FALSE;
	Enable		: BOOL;
	boolbuf1		: BOOL;
	boolbuf2		: BOOL;
END_STRUCT
END_TYPE

// ---- Data types/ST_OneLineAir.TcDUT
TYPE ST_OneLineAir :
STRUCT
	Air	: ARRAY [1..AirNo] OF INT;
END_STRUCT
END_TYPE

// ---- Data types/ST_OneLineTable.TcDUT
TYPE ST_OneLineTable :
STRUCT
	Dist		: ARRAY [1..No] OF LREAL;
	Velocity   : ARRAY [1..No] OF LREAL;
	Acc		: ARRAY [1..No] OF LREAL;
	Dec		: ARRAY [1..No] OF LREAL;
	Jerk		: ARRAY [1..No] OF LREAL;
	Delay	: LREAL;
END_STRUCT
END_TYPE

// ---- Data types/ST_ProAndManRelativeState.TcDUT
TYPE ST_ProAndManRelativeState :
STRUCT
	ErrorID 				: ARRAY [1..2] OF UDINT;
	Done 				: ARRAY [1..2] OF BOOL;
	Busy 				: ARRAY [1..2] OF BOOL;
	Active 				: ARRAY [1..2] OF BOOL;
	CommandAborted 	: ARRAY [1..2] OF BOOL;
	Error 				: ARRAY [1..2] OF BOOL;
END_STRUCT
END_TYPE

// ---- Data types/ST_Produce.TcDUT
TYPE ST_Produce :
STRUCT
	Start				: ARRAY [0..MAX_ARRAY] OF LREAL :=[0,MAX_ARRAY(0)] ;
	End				: ARRAY [0..MAX_ARRAY] OF LREAL :=[0,MAX_ARRAY(0)];
	Dist				: ARRAY [0..MAX_ARRAY] OF LREAL :=[0,MAX_ARRAY(0)];
	Velocity			: ARRAY [0..MAX_ARRAY] OF LREAL :=[0,MAX_ARRAY(0)];
	TPhase1			: ARRAY [0..MAX_ARRAY] OF LREAL :=[0,MAX_ARRAY(0)];
	TPhase2			: ARRAY [0..MAX_ARRAY] OF LREAL :=[0,MAX_ARRAY(0)];
	Acceleration		: ARRAY [0..MAX_ARRAY] OF LREAL :=[0,MAX_ARRAY(0)];
	Deceleration		: ARRAY [0..MAX_ARRAY] OF LREAL :=[0,MAX_ARRAY(0)];
	Jerk				: ARRAY [0..MAX_ARRAY] OF LREAL :=[0,MAX_ARRAY(0)];
END_STRUCT
END_TYPE

// ---- Data types/ST_RingBuffer.TcDUT
TYPE ST_RingBuffer :
STRUCT
	Table		: ARRAY [0..3599] OF LREAL;
END_STRUCT
END_TYPE

// ---- Data types/ST_RingBufferIO.TcDUT
TYPE ST_RingBufferIO :
STRUCT
	Table		: ARRAY [0..3599] OF BOOL;
END_STRUCT
END_TYPE

// ---- Data types/ST_RingBufferIOPart.TcDUT
TYPE ST_RingBufferIOPart :
STRUCT
	(*200當確認點、是否傳送到*)
	Table	: ARRAY [0..200] OF BOOL;
END_STRUCT
END_TYPE

// ---- Data types/ST_RingBufferPart.TcDUT
TYPE ST_RingBufferPart :
STRUCT
	(*200當確認點、是否傳送到*)
	Table	: ARRAY [0..200] OF LREAL;
END_STRUCT
END_TYPE

// ---- Data types/ST_SetPosByUI.TcDUT
TYPE ST_SetPosByUI :
STRUCT
	Position	:LREAL:=0;
	Axis		:INT:=1;
	Execute	:BOOL:=FALSE;
END_STRUCT
END_TYPE

// ---- Data types/ST_SlaveEcData.TcDUT
TYPE ST_SlaveEcData :
STRUCT
	Name	: STRING(31);
	sType   : STRING(15);
	InfoData: UINT;
	PortA	: UDINT;
	PortB	: UDINT;
	PortC	: UDINT;
	PortD	: UDINT;
END_STRUCT
END_TYPE

// ---- Data types/ST_SubProgramConfig.TcDUT
TYPE ST_SubProgramConfig :
STRUCT
	Reaction 		: INT;
	TotalTableSIze 	: DINT;
	StartIdx			: DINT;
	EndIdx			: DINT;
END_STRUCT
END_TYPE

// ---- Data types/ST_SubProgramTable.TcDUT
TYPE ST_SubProgramTable :
STRUCT
	AxisTable						: ARRAY [1..No, 0..59999] OF LREAL;
	AirTable							: ARRAY [1..AirNo, 0..59999] OF BOOL;
	ExFSpdUpTable					: ARRAY [0..59999] OF BOOL;
END_STRUCT
END_TYPE

// ---- Data types/ST_Touch.TcDUT
TYPE ST_Touch :
STRUCT
	TouchTime		: UDINT;
	CurTime			: UDINT;
	Enable			: BOOL;
	Miss			: BOOL;
	boolbuf1			: BOOL;
	boolbuf2			: BOOL;
	boolbuf3			: BOOL;
	boolbuf4			: BOOL;
	boolbuf5			: BOOL;
	boolbuf6			: BOOL;
END_STRUCT
END_TYPE

// ---- Data types/ST_TouchAdjustConfig.TcDUT
TYPE ST_TouchAdjustConfig :
STRUCT
    pAxis           : INT;
    TouchNo         : INT;
    UpBound         : REAL;
    DownBound       : REAL;
    RangeUp         : REAL; 
    RangeDown       : REAL;
    UpCountLimit    : REAL; (* + *)
    DownCountLimit  : REAL; (* - *)
    TouchStartIdx   : DINT;
    TouchEndIdx     : DINT;
    AdjustStartIdx  : DINT;
    AdjustEndIdx    : DINT;
    Enable          : BOOL;
END_STRUCT
END_TYPE

// ---- Data types/ST_TouchConfig.TcDUT
TYPE ST_TouchConfig :
STRUCT
	StartIdx		: ARRAY[0..999] OF DINT;
	EndIdx		: ARRAY[0..999] OF DINT;
END_STRUCT
END_TYPE

// ---- Data types/ST_TouchProbe.TcDUT
TYPE ST_TouchProbe :
STRUCT
	Execute			: BOOL:=FALSE;
	WindowOnly		: BOOL:=FALSE;
	FirstPosition		: LREAL:=0;
	LastPosition 		: LREAL:=0;
	Trigger_Ref	         : TRIGGER_REF ;

	RecordPosition	: LREAL;
END_STRUCT
END_TYPE

// ---- Data types/ST_TouchProbeHomeByUI.TcDUT
TYPE ST_TouchProbeHomeByUI :
STRUCT
	ZRTSpeed		: LREAL;
	ZRTSet			: LREAL;
	Execute			: BOOL;
	boolbuf1			: BOOL;
	boolbuf2			: BOOL;
	boolbuf3			: BOOL;
	boolbuf4			: BOOL;
	boolbuf5			: BOOL;
	boolbuf6			: BOOL;
	boolbuf7			: BOOL;
END_STRUCT
END_TYPE

// ---- Data types/ST_TouchTableBuf.TcDUT
TYPE ST_TouchTableBuf :
STRUCT
	Table	: ARRAY [1..TouchNo, 0..1999] OF BOOL;
	OK		: BOOL;
END_STRUCT
END_TYPE

// ---- Global Variables/ENUMSTATE.TcDUT
{attribute 'qualified_only'}
{attribute 'strict'}
TYPE 
	ENUMSTATE 						: (S_AUTO, S_TEST, S_MPG, S_MANMOV, S_ZRT, S_IDLE, S_ERROR, S_TROUBLESHOOT, S_TROSHO_MANMOV);
END_TYPE

// ---- Global Variables/MachineSubTypeEnum.TcDUT
{attribute 'qualified_only'}
{attribute 'strict'}
TYPE 
	MachineSubTypeEnum				: (None, CE);
END_TYPE

// ---- Global Variables/MachineTypeEnum.TcDUT
{attribute 'qualified_only'}
{attribute 'strict'}
TYPE 
	MachineTypeEnum					: (_08x, _25x, _42x, _60x, _1020, _1320, _1350, _1320XYZ, _1370XYZ);
END_TYPE

// ---- Global Variables/MANMOVEENUM.TcDUT
{attribute 'qualified_only'}
{attribute 'strict'}
TYPE 
	MANMOVEENUM	: (S_MANINITIAL, S_MANMOVE, S_MOVESTOP);
END_TYPE

// ---- Global Variables/MotorVenderEnum.TcDUT
{attribute 'qualified_only'}
{attribute 'strict'}
TYPE 
	MotorVenderEnum					: (SANYO, DELTA, YASKAWA);
END_TYPE

// ---- Global Variables/Global_Variables.TcGVL
{attribute 'Tc2GvlVarNames'}
VAR_GLOBAL
	SoftVersion 					: STRING := '1.5.3';
	PLC_StartRunning				: BOOL:=FALSE;
	State							: INT:=ENUMSTATE.S_IDLE;
	AmsNetId						: T_AmsNetId := '0.0.0.0.2.1'; (* NetId of EtherCAT Master *)
	DeviceNetId               		: T_AmsNetId;
	MotorVendor						: INT;
	MachineType						: INT;
	MachineSubType					: INT;
	FServoOn						: BOOL;
	FAlarmReset						: BOOL;
	AirIsOpen						: ARRAY [1..AirNo] OF BOOL;
	Oil								: ARRAY [1..OilNo] OF ST_OIL;
	LightOGR						: ARRAY [1..3] OF BOOL;
	Touch							: ARRAY [1..TouchNo] OF ST_Touch;
	TouchMissStop					: BOOL:=FALSE;
	CounterSwitch					: BOOL;
	NoMaterialEnable				: BOOL;
	PressDetect						: BOOL;
	Inputstate						: ST_Inputstate;
	Producing						: BOOL:=FALSE;
    SubRunning  					: BOOL;
    SubRunAloneFirstTime   			: BOOL:=TRUE;
	MoveToColPosRunning 			: BOOL:=FALSE;
	MoveToPosFirstTime 				: BOOL:=TRUE;
	CycleLastCmdIsRun				: BOOL:= TRUE;
	ProFirstTime					: BOOL:=TRUE;
	ZRTFirstTime					: BOOL:=TRUE;
	Emgstoptrig						: BOOL:=FALSE;
	Override						: LREAL;(*0 ~ 100.0*)
	IsUseVROverride					: BOOL;
	IsVirtualOOverride				: BOOL;
	SpeedDownTo0					: BOOL;
	Mpg_PositiveMove				: BOOL;
	Mpg_NegativeMove				: BOOL;
	Master							: ST_McFBInOutVar;
	Axis								: ARRAY [1..No] OF ST_McFBInOutVar;
	AxisIsOn							: ARRAY [1..No] OF BOOL;
	AxisValue						: ARRAY [1..No] OF ST_McValue;
	AxisProduce 						: ARRAY [1..No] OF ST_Produce;
	AxisManMove					: ARRAY [1..No] OF ST_ManMove;
	AxisHoming AT %Q* 				: ARRAY [1..No] OF  ST_Homing;
	AxisOpMode	AT%Q*				: ARRAY [1..No] OF SINT:=[No(8)];
	DigOutSlave AT %Q*  		         		 : ARRAY [1..DigOutSlaveNum] OF ST_DigitOutput;
	AxisTouchProbe					 : ARRAY [1..No] OF ST_TouchProbe;
	TouchProbeFunction AT%Q*     	   	: ARRAY [1..No] OF UINT:=[No(15)];
	DigInSlave AT %I*   				: ARRAY [1..DigInSlaveNum] OF ST_DigitInput;
	AnaInSlave AT%I*					: ARRAY [1..AnaInSlaveNum] OF ST_AnaInput;
	EL5101SlaveValue AT%I*			: UINT;
	EL3062_VR AT%I*					: INT;
	MasterAxis						: ST_MasterAxisValue;
	MasterAxisPos					: ST_MasterAxisPos;
	AxisCountPosByInput	AT %I*		: ARRAY [1..No] OF DINT;
	SetAxisPosByCountPos			: ARRAY [1..No] OF BOOL;
	UISetPosAllComplete				: BOOL:=FALSE;
	FeederNo						: INT;
	RotateWNo						: INT;
	RWAddFeederRatio				: REAL;
	ProAndManRelative				: ARRAY [1..No] OF ST_ProAndManRelativeState;
	CurManMovAxis   					: INT;
	Cam							: ARRAY [1..No] OF ST_Cam;
	CamTable1						: ARRAY [1..No] OF ST_CamTable;
	CamTable2						: ARRAY [1..No] OF ST_CamTable;
	OneLineTable					: ARRAY [1..MAX_ARRAY] OF ST_OneLineTable;
	OneLineAir						: ARRAY [1..MAX_ARRAY] OF ST_OneLineAir;
	OneLineLineNum					: DINT;
	Halt								: ARRAY [1..No] OF MC_Halt;
	BrakeParam						: ARRAY [1..No] OF ST_BrakeParam;
	BigPowerSwitch					: BOOL;
	DriveAlarmCode AT %I*			: ARRAY [1..No] OF ST_DriveAlarmCode;
	BuzzerIsOpen						: BOOL:=FALSE;
	ExFeederSpeedUp				: BOOL:=FALSE;
	AlarmList							: ST_InputState;
	SaftyOn							: BOOL;
	IOSwitch						: ST_IOSwitch;
	IsZrtGrpSelect					: BOOL:=FALSE;

	RingBuffer						: ARRAY [1..No] OF ST_RingBuffer;
	RingBufferPart					: ARRAY [1..No] OF ST_RingBufferPart;
	RingBufferAir						: ARRAY [1..AirNo] OF ST_RingBufferIO;
	RingBufferAirPart					: ARRAY [1..AirNo] OF ST_RingBufferIOPart;
	RingBufferTouch					: ARRAY [1..TouchNo] OF ST_RingBufferIO;
	RingBufferTouchPart				: ARRAY [1..TouchNo] OF ST_RingBufferIOPart;
	RingBufferExFeederSpeedUp		: ST_RingBufferIO;
	RingBufferExFeederSpeedUpPart	: ST_RingBufferIOPart;
	RingBufferAxesPosBuf            : ARRAY [1..No] OF ST_AxisPosBuf;
	RingBufferAxesVelBuf            : ARRAY [1..No] OF ST_AxisVelBuf;
	RingBufferAxesTrqBuf            : ARRAY [1..No] OF ST_AxisTrqBuf;


	IsGetTableBuf					: BOOL;
	AxisTableBuf						: ST_AxisTableBuf;
	TouchTableBuf					: ST_TouchTableBuf;
	AirTableBuf						: ST_AirTableBuf;
	ExFSpdUpTableBuf				: ST_ExFSpdUpTableBuf;

	AxisTable1						: ARRAY [1..No, 0..299999] OF LREAL;
	AxisTable2						: ARRAY [1..No, 0..299999] OF LREAL;
	TouchTable						: ARRAY [1..TouchNo, 0..299999] OF BOOL;
	AirTable							: ARRAY [1..AirNo, 0..299999] OF BOOL;
	ExFSpdUpTable					: ARRAY [0..299999] OF BOOL;

	TouchAdjustTable				: ARRAY [1..TouchAdjustNo, 0..119999] OF LREAL;
	TouchAdjustConfig				: ARRAY [1..TouchAdjustNo] OF ST_TouchAdjustConfig;

	SubProgramConfig				: ARRAY [1..SubProgramNo] OF ST_SubProgramConfig;
	SubProgramTable				: ARRAY [1..SubProgramNo] OF ST_SubProgramTable;

	(* EtherCAT *)
    SlaveConfigData 				: ARRAY [0..MaxSlaves] OF ST_EcSlaveConfigData;		
	SlaveEcData						: ARRAY [0..MaxSlaves] OF ST_SlaveEcData;
	SlaveEcInfoData AT%I*			: ARRAY [0..MaxSlaves] OF UINT;

	AxesUseModulo					: ARRAY [1..No] OF BOOL;
	AxesModuloTurns					: ARRAY [1..No] OF DINT;
	AxesGradPerTurn					: ARRAY [1..No] OF DINT;
	AxesModuloOGrad				: ARRAY [1..No] OF LREAL;
	AxesTorque AT %I*				:ARRAY [1..NO] OF INT;

	(* PowerOff 功能*)	
	PLCToUIShutDown					:BOOL;
	InPowerOffProcess				:BOOL;
	PowerOffCnt						:INT;

	AlarmListClear					:BOOL;
	RoutinCheck						: BOOL;
	IsConnecting					: BOOL := TRUE;
	IsDebugMode						: BOOL := FALSE;

END_VAR
VAR_GLOBAL CONSTANT
	No				: INT:=20;
	OilNo			: INT:=1;
	AirNo			: INT:=12;
	TouchNo		: INT:=4;
	TimerNo			: INT:=3;
	DigOutSlaveNum   : INT:=3;
	DigInSlaveNum	: INT:=4;
	AnaInSlaveNum	: INT:=1;
	MAX_ARRAY		: INT:=100;
	SubProgramNo	: INT:=10;
	G5ConfigNo		: INT:=10;
	MaxSlaves		: INT:=99;
	TouchAdjustNo   : INT:=4;
END_VAR

// ---- Global Variables/Variable_Configuration.TcGVL
{attribute 'Tc2GvlVarNames'}
VAR_CONFIG
END_VAR

// ---- POUs/MAIN.TcPOU
PROGRAM MAIN
VAR
	ENUM 			:(S_PLCINITIAL, S_PLC_BigPowerOn, S_PLC_FSetPos, S_PLC_START);
	PLCState		: INT;
	idx 				: INT;
	Trig				: R_TRIG;
	Count1			: INT:=0;
	Timer			: TON;
	GetMachineInfo      :FB_GetMachineInfo;
	FSetPosExe		:BOOL;
END_VAR

IF PLC_StartRunning = TRUE THEN
	CASE PLCState OF
		S_PLCINITIAL:(*初始*)
			GetMachineInfo(Execute:= TRUE);
			IF NOT GetMachineInfo.Busy THEN
				GetMachineInfo.Execute := FALSE;
				PLCState := S_PLC_BigPowerOn;
			END_IF

		S_PLC_BigPowerOn:
			BigPowerSwitch := TRUE;
						IOMapping();
			Timer(IN:= TRUE,PT:= T#500ms );
			IF Timer.Q THEN
				Timer(IN:= FALSE);
				FSetPosExe := TRUE;
				PLCState := S_PLC_FSetPos;
			END_IF
		S_PLC_FSetPos:
						prAxis();
			Axis[1].fbMC_SetPosition(
				Execute	:=FSetPosExe,
				Position	:= 0,
				Axis		:= Axis[1].Axis
			);
			IF Axis[1].fbMC_SetPosition.Done THEN
				FSetPosExe := FALSE;
				Timer(IN:= TRUE,PT:= T#1000ms );
			END_IF
			Timer();
			IF Timer.Q THEN
				Timer(IN:= FALSE);
				PLCState := S_PLC_START;
			END_IF
		S_PLC_START:

						IOMapping();
						CommunicationQualityCheck();

						EMGStop();
						Error();

						SetCountPosToActPos();
						prAxis();

			FServoOn:=TRUE;

						Mpg();
						SetOverride();

						Produce();
						SubRunAlone();
						MoveToColPos();
						ManMove();
						HomeByTouchProbe();
						SetPosByUI();
						MCRelativeMove();

						AlertLight();

						IOMapping();
						AxisStatusDataStore();
						EncoderClear();
						UPS();
	END_CASE

END_IF

END_PROGRAM

// ---- POUs/FB/FB_GetMachineInfo.TcPOU
FUNCTION_BLOCK FB_GetMachineInfo
VAR_INPUT
	Execute	:BOOL;
END_VAR
VAR_OUTPUT
	Busy	:BOOL;
END_VAR
VAR
	seq						:INT:=0;
	idx						:INT:=0;

	fbGetLocalAmsNetId 		:FB_GetLocalAmsNetId;
	addrBytes				:AMSNETID :=[ 0,0,0,0,0,0];(* TwinCAT-specific network address as array of byte *)

	iofGetDeviceNetId 		:IOF_GetDeviceNetId;

 	fbEcGetAllSlaveAddr 		:FB_EcGetAllSlaveAddr;
    	slaveAddr          			:ARRAY[0..MaxSlaves] OF UINT;

	fbEcGetConfSlaves 		:FB_EcGetConfSlaves;

	vendorId 	: UDINT;
END_VAR

IF Execute THEN
	Busy := TRUE;

	CASE seq OF
		0:
			fbGetLocalAmsNetId(
				bExecute :=TRUE,
				tTimeOut := t#2s,
				AddrString =>AmsNetId,
				AddrBytes =>AddrBytes,
			);

			IF NOT fbGetLocalAmsNetId.bBusy THEN
				fbGetLocalAmsNetId(bExecute := FALSE);
				seq := 1;
			END_IF
		1:
			iofGetDeviceNetId(
				NetID := AmsNetId,
				Start := TRUE,
				DeviceID := 1,
				DeviceNetId =>DeviceNetId,
			);

			IF NOT iofGetDeviceNetId.BUSY THEN
				iofGetDeviceNetId(Start := FALSE);
				seq		       := 2;
			END_IF
		2:
			fbEcGetAllSlaveAddr(
				sNetId:= DeviceNetId,
				pAddrBuf:= ADR(slaveAddr),
				cbBufLen:= SIZEOF(slaveAddr[0]) * (MaxSlaves + 1),
				bExecute:= TRUE,
				tTimeout:= ,
				bBusy=> ,
				bError=> ,
				nErrId=> ,
				nSlaves=> );
			IF NOT fbEcGetAllSlaveAddr.bBusy THEN
				fbEcGetAllSlaveAddr(bExecute:= FALSE);
				seq       := 3;
			END_IF

		3:
			fbEcGetConfSlaves(
				sNetId:= DeviceNetId,
				pArrEcConfSlaveInfo:= ADR(SlaveConfigData),
				cbBufLen:= SIZEOF(SlaveConfigData[0]) * (MaxSlaves + 1),
				bExecute:= TRUE,
				tTimeout:= ,
				bBusy=> ,
				bError=> ,
				nErrorId=> ,
				nSlaves=> );
			IF NOT fbEcGetConfSlaves.bBusy THEN
				FOR idx := 0 TO MaxSlaves DO
					SlaveEcData[idx].Name := SlaveConfigData[idx].sName;
					SlaveEcData[idx].sType := SlaveConfigData[idx].sType;
				END_FOR
				fbEcGetConfSlaves(bExecute:= FALSE);
				seq       := 4;
			END_IF
		4:
			Axis[1].fbSDORead(
				bExecute:=TRUE,
				sNetId:= DeviceNetId,
				nSlaveAddr :=1009,(*第一軸*)
				nIndex:=16#1018,
				nSubIndex :=1,
				 pDstBuf:= ADR(vendorId),
				cbBufLen:=SIZEOF(vendorId)
			);
			IF NOT Axis[1].fbSDORead.bBusy THEN
				 Axis[1].fbSDORead.bExecute := FALSE;
				seq		       := 5;

				IF vendorId = 16#01DD THEN
					MotorVendor := MotorVenderEnum.DELTA;
				ELSIF vendorId = 16#0539 THEN
					MotorVendor := MotorVenderEnum.YASKAWA;
				ELSE
					MotorVendor := MotorVenderEnum.SANYO;
				END_IF
			END_IF
		5:
			Busy:=FALSE;

	END_CASE
END_IF

END_FUNCTION_BLOCK

// ---- POUs/IOMapping.TcPOU
PROGRAM IOMapping
VAR
	idx						: INT:=1;
	Outputidx1				: INT:=1;
	Outputidx2				: INT:=1;
	NormalCtrlPowerOffTimer	: TON;
	ForceCtrlPowerOffTimer	: TON;
	UIShutDownTimer  		: TON;
	CtrlPowerOffTimer 		: TON;
	PowerOffLCnt			: INT;
	ForceCtrlPowerOff		: BOOL;
	NormalCtrlPowerOff		: BOOL;
	CheckTimer				: TON;
END_VAR

(*-----------------------------------Output1------------------------------------*)
(*三色警示燈*)
DigOutSlave[1].Output[1] := LightOGR[1];
DigOutSlave[1].Output[2] := LightOGR[2];
(*大電開關*)
DigOutSlave[1].Output[3] := BigPowerSwitch;
(*線架加速*)
DigOutSlave[1].Output[4] := ExFeederSpeedUp;
(*蜂鳴器*)
DigOutSlave[1].Output[5] := BuzzerIsOpen;
(*油機*)
DigOutSlave[1].Output[6] := Oil[1].IsOpen;
(*DigOutSlave[1].Output[7]:=;*)
DigOutSlave[1].Output[8] := ForceCtrlPowerOff OR NormalCtrlPowerOff;
DigOutSlave[1].Output[9] := LightOGR[3];

(*-----------------------------------Output2------------------------------------*)
(*汽缸*)
DigOutSlave[2].Output[1] := AirIsOpen[1];
DigOutSlave[2].Output[2] := AirIsOpen[2];
DigOutSlave[2].Output[3] := AirIsOpen[3];
DigOutSlave[2].Output[4] := AirIsOpen[4];
DigOutSlave[2].Output[5] := AirIsOpen[5];
DigOutSlave[2].Output[6] := AirIsOpen[6];
DigOutSlave[2].Output[7] := AirIsOpen[7];
DigOutSlave[2].Output[8] := AirIsOpen[8];
DigOutSlave[2].Output[9] := AirIsOpen[9];
DigOutSlave[2].Output[10] := AirIsOpen[10];
DigOutSlave[2].Output[11] := AirIsOpen[11];
DigOutSlave[2].Output[12] := AirIsOpen[12];
DigOutSlave[2].Output[13] := FAlarmReset;
(*DigOutSlave[2].Output[14] := *)
DigOutSlave[2].Output[15] := FServoOn;

(*-----------------------------------Output3------------------------------------*)
DigOutSlave[3].Output[1] := IOSwitch.SafetyLockDisable;
(*
DigOutSlave[3].Output[2] := 
DigOutSlave[3].Output[3] := 
DigOutSlave[3].Output[4] := 
DigOutSlave[3].Output[5] := 
DigOutSlave[3].Output[6] := 
DigOutSlave[3].Output[7] := 
DigOutSlave[3].Output[8] := 
DigOutSlave[3].Output[9] := 
DigOutSlave[3].Output[10] :=
DigOutSlave[3].Output[11] :=
DigOutSlave[3].Output[12] :=
DigOutSlave[3].Output[13] :=
DigOutSlave[3].Output[14] :=
DigOutSlave[3].Output[15] :=
*)

(*-------------------------------------Input1--------------------------------------*)
Inputstate.PowerOff   		 :=  DigInSlave[1].Input[1];
Inputstate.Reset			 :=  DigInSlave[1].Input[2];
Inputstate.Producing		 :=  DigInSlave[1].Input[3];
Inputstate.Testing			 :=  DigInSlave[1].Input[4];
Inputstate.EditLock		 	 :=  DigInSlave[1].Input[5];
Inputstate.ExFeederError	 :=  DigInSlave[1].Input[6];
Inputstate.SafetyError		 :=  DigInSlave[1].Input[7];
Inputstate.OilError			 :=  DigInSlave[1].Input[8];
Inputstate.VRSwitch		 	 :=  DigInSlave[1].Input[9];
Inputstate.EMGStop		 	 :=  DigInSlave[1].Input[10];
Inputstate.HomeA			 :=  DigInSlave[1].Input[11];
Inputstate.plusA			 :=  DigInSlave[1].Input[12];
Inputstate.negA			 	 :=  DigInSlave[1].Input[13];
Inputstate.plusY			 :=  DigInSlave[1].Input[14];
Inputstate.negY				 :=  DigInSlave[1].Input[15];
Inputstate.SW				 :=  DigInSlave[1].Input[16];


(*-------------------------------------Input2--------------------------------------*)
Inputstate.Touch1   		 :=  DigInSlave[2].Input[1];
Inputstate.Touch2			 :=  DigInSlave[2].Input[2];
Inputstate.Touch3			 :=  DigInSlave[2].Input[3];
Inputstate.Touch4			 :=  DigInSlave[2].Input[4];
Inputstate.StopCycle		 :=  DigInSlave[2].Input[5];
Inputstate.ExDeviceError	 :=  DigInSlave[2].Input[6];

Inputstate.FAlarm_1370		 := DigInSlave[2].Input[9];
Inputstate.PowerBit1		 := DigInSlave[2].Input[10];
Inputstate.PowerBit0		 := DigInSlave[2].Input[11];

Inputstate.ChoiceAxisBit4	 := DigInSlave[2].Input[12];
Inputstate.ChoiceAxisBit3	 := DigInSlave[2].Input[13];
Inputstate.ChoiceAxisBit2	 := DigInSlave[2].Input[14];
Inputstate.ChoiceAxisBit1	 := DigInSlave[2].Input[15];
Inputstate.ChoiceAxisBit0	 := DigInSlave[2].Input[16];

(*-------------------------------------Input3--------------------------------------*)
Inputstate.NG		   		 :=  DigInSlave[3].Input[1];
Inputstate.Mpg_PositiveBtn	 :=  DigInSlave[3].Input[2];
Inputstate.Mpg_NegativeBtn	 :=  DigInSlave[3].Input[3];
Inputstate.Zrt				 :=  DigInSlave[3].Input[4];

(*:=  DigInSlave[3].Input[5];
:=  DigInSlave[3].Input[4];
:=  DigInSlave[3].Input[5];
:=  DigInSlave[3].Input[6];
:=  DigInSlave[3].Input[7];
:=  DigInSlave[3].Input[8];
:=  DigInSlave[3].Input[9];
:=  DigInSlave[3].Input[10];
:=  DigInSlave[3].Input[11];
:=  DigInSlave[3].Input[12];
:=  DigInSlave[3].Input[13];
:=  DigInSlave[3].Input[14];
:=  DigInSlave[3].Input[15];
:=  DigInSlave[3].Input[16];
*)

(*-------------------------------------Input4--------------------------------------*)
IF MachineSubType = MachineSubTypeEnum.CE THEN
	Inputstate.SafetyError1   	 := DigInSlave[4].Input[1];
	Inputstate.SafetyError2		 := DigInSlave[4].Input[2];
	Inputstate.SafetyError3		 := DigInSlave[4].Input[3];
	Inputstate.SafetyError4		 := DigInSlave[4].Input[4];
	Inputstate.FrontEStop		 := DigInSlave[4].Input[5];
	Inputstate.SideEStop	     := DigInSlave[4].Input[6];
	Inputstate.RearEStop		 := DigInSlave[4].Input[7];
	Inputstate.DecoilorEStop	 := DigInSlave[4].Input[8];
END_IF
(*
 :=  DigInSlave[4].Input[9];
 :=  DigInSlave[4].Input[10];
 :=  DigInSlave[4].Input[11];
 :=  DigInSlave[4].Input[12];
 :=  DigInSlave[4].Input[13];
 :=  DigInSlave[4].Input[14];
 :=  DigInSlave[4].Input[15];
 :=  DigInSlave[4].Input[16];
 *)

(*--------------------------PowerOff--------------------------------*)
PowerOffFunc();
(*--------------------------ConnectionCheck--------------------------------*)
ConnectionCheck();
(*--------------------------LatchAlarmInput--------------------------------*)
LatchAlarmInput();

ACTION ConnectionCheck:
IF NOT IsDebugMode THEN
    CheckTimer(IN:= TRUE, PT:= T#5s);
    IF IsConnecting THEN
        IF RoutinCheck THEN
            CheckTimer(IN:= FALSE);
            RoutinCheck := FALSE;
        ELSE
            IF CheckTimer.Q THEN
                IsConnecting := FALSE;
            END_IF
        END_IF
    END_IF
ELSE
	CheckTimer(IN:= FALSE);
END_IF
END_ACTION

ACTION LatchAlarmInput:
AlarmList.Reset         := NOT AlarmListClear AND SEL(Inputstate.Reset , AlarmList.Reset, TRUE);
AlarmList.OilError      := NOT AlarmListClear AND SEL(Inputstate.OilError , AlarmList.OilError, TRUE);
AlarmList.EMGStop       := NOT AlarmListClear AND SEL(Inputstate.EMGStop , AlarmList.EMGStop, TRUE);
AlarmList.FAlarm_1370   := NOT AlarmListClear AND SEL(Inputstate.FAlarm_1370 , AlarmList.FAlarm_1370, TRUE);
AlarmList.ExDeviceError := NOT AlarmListClear AND SEL(Inputstate.ExDeviceError , AlarmList.ExDeviceError, TRUE);

AlarmList.NG            := NOT AlarmListClear AND SEL(Inputstate.NG     , AlarmList.NG, TRUE);

AlarmList.SafetyError   := NOT AlarmListClear AND SEL(Inputstate.SafetyError  AND IOSwitch.SaftyEnable AND State <> ENUMSTATE.S_AUTO AND State <> ENUMSTATE.S_TEST AND State <> ENUMSTATE.S_MPG, AlarmList.SafetyError, TRUE);
AlarmList.SafetyError1  := NOT AlarmListClear AND SEL(Inputstate.SafetyError1 AND IOSwitch.SaftyEnable AND State <> ENUMSTATE.S_AUTO AND State <> ENUMSTATE.S_TEST AND State <> ENUMSTATE.S_MPG, AlarmList.SafetyError1, TRUE);
AlarmList.SafetyError2  := NOT AlarmListClear AND SEL(Inputstate.SafetyError2 AND IOSwitch.SaftyEnable AND State <> ENUMSTATE.S_AUTO AND State <> ENUMSTATE.S_TEST AND State <> ENUMSTATE.S_MPG, AlarmList.SafetyError2, TRUE);
AlarmList.SafetyError3  := NOT AlarmListClear AND SEL(Inputstate.SafetyError3 AND IOSwitch.SaftyEnable AND State <> ENUMSTATE.S_AUTO AND State <> ENUMSTATE.S_TEST AND State <> ENUMSTATE.S_MPG, AlarmList.SafetyError3, TRUE);
AlarmList.SafetyError4  := NOT AlarmListClear AND SEL(Inputstate.SafetyError4 AND IOSwitch.SaftyEnable AND State <> ENUMSTATE.S_AUTO AND State <> ENUMSTATE.S_TEST AND State <> ENUMSTATE.S_MPG, AlarmList.SafetyError4, TRUE);

AlarmList.PanelEStop    := NOT AlarmListClear AND SEL(Inputstate.PanelEStop     , AlarmList.PanelEStop, TRUE);
AlarmList.FrontEStop    := NOT AlarmListClear AND SEL(Inputstate.FrontEStop     , AlarmList.FrontEStop, TRUE);
AlarmList.SideEStop     := NOT AlarmListClear AND SEL(Inputstate.SideEStop      , AlarmList.SideEStop, TRUE);
AlarmList.RearEStop     := NOT AlarmListClear AND SEL(Inputstate.RearEStop      , AlarmList.RearEStop, TRUE);
AlarmList.DecoilorEStop := NOT AlarmListClear AND SEL(Inputstate.DecoilorEStop  , AlarmList.DecoilorEStop, TRUE);

AlarmList.ExFeederError := NOT AlarmListClear AND SEL(Inputstate.ExFeederError AND State <> ENUMSTATE.S_AUTO AND State <> ENUMSTATE.S_TEST AND State <> ENUMSTATE.S_MPG, AlarmList.ExFeederError, TRUE);


AlarmListClear := FALSE;
END_ACTION

ACTION PowerOffFunc:
IF Inputstate.PowerOff THEN
	NormalCtrlPowerOffTimer(IN:= TRUE,PT:= T#200ms );
	ForceCtrlPowerOffTimer(IN:= TRUE,PT:= T#3000ms );
	IF ForceCtrlPowerOffTimer.Q THEN
        BigPowerSwitch    :=FALSE;
		InPowerOffProcess :=TRUE;
		ForceCtrlPowerOff :=TRUE;
	END_IF
ELSE
	IF NormalCtrlPowerOffTimer.Q THEN
		InPowerOffProcess := TRUE;
	END_IF

	IF  InPowerOffProcess THEN

		BigPowerSwitch :=FALSE;    	
		UIShutDownTimer(IN:= TRUE, PT:= T#1000ms);

		IF UIShutDownTimer.Q THEN
			PLCToUIShutDown := TRUE;

			IF PowerOffCnt <> PowerOffLCnt THEN
				PowerOffLCnt := PowerOffCnt;				
			ELSIF PowerOffCnt = PowerOffLCnt THEN
				CtrlPowerOffTimer(IN:= TRUE,PT:= T#1000ms );
				IF CtrlPowerOffTimer.Q THEN
					NormalCtrlPowerOff :=TRUE;
				END_IF
			END_IF

		END_IF
	ELSE
		BigPowerSwitch	   :=TRUE;
		PLCToUIShutDown	   :=FALSE;
		NormalCtrlPowerOff :=FALSE;
		ForceCtrlPowerOff  :=FALSE;
		UIShutDownTimer(IN:= FALSE);
		CtrlPowerOffTimer(IN:= FALSE);
	END_IF
	NormalCtrlPowerOffTimer(IN:= FALSE);
	ForceCtrlPowerOffTimer(IN:= FALSE);
END_IF
END_ACTION

END_PROGRAM

// ---- POUs/EMGStop.TcPOU
PROGRAM EMGStop
VAR
	ENUMSTOPSTATE :(S_DisableSetPointGenerator ,S_STOP_DECOUPLE, S_STOP_HALT, S_STOP_RESET, S_STOP_RELATIVE, S_STOP_IDLE);
	FirstTime		: BOOL:=TRUE;
	EMGStopState	: ARRAY [1..No] OF INT;
	idx				: INT:=1;
	MasterResetTrig	: R_TRIG;
	HaltTrig			   : ARRAY [1..No] OF R_TRIG;
	ResetTrig		: ARRAY [1..No] OF R_TRIG;
	ResetTimer		: TON;
	RelativeMOVE	: RelativeMOVE;
	RelativeMOVE2	: RelativeMOVE2;
	EMGStopCompleteNum : INT:=0;
	CloseOil			: FB_CloseOil;
END_VAR



IF Emgstoptrig = TRUE THEN
	IF FirstTime THEN
		FirstTime	:= FALSE;
		IF State <> ENUMSTATE.S_ERROR AND State <> ENUMSTATE.S_TROUBLESHOOT AND State <> ENUMSTATE.S_TROSHO_MANMOV THEN
			State:= ENUMSTATE.S_IDLE;
		END_IF
		ProFirstTime   := TRUE;
		SubRunAloneFirstTime := TRUE;
		MoveToPosFirstTime	:= TRUE;
		ZRTFirstTime := TRUE;
		SubRunning	:= FALSE;
		MoveToColPosRunning := FALSE;
				CloseOil();(*關閉油機*)
		SpeedDownTo0 := FALSE;


		(*---------- 生產部分---------*)
(*		Override		 := 100;*)
		Producing 	 := FALSE;
		CycleLastCmdIsRun := TRUE;
		(*--------------------------------*)

		MasterResetTrig(CLK:= FALSE);
		FOR idx:=1 TO No DO
			EMGStopState[idx] := S_DisableSetPointGenerator;
			HaltTrig[idx](CLK:=FALSE);
			ResetTrig[idx](CLK:= FALSE);
		END_FOR
	END_IF

(*Master Reset*)
MasterResetTrig(CLK:= TRUE);
Master.fbMC_Reset(
	Execute:=MasterResetTrig.Q,
	Axis:=Master.Axis
);
Master.fbMC_MoveRelative[1](
	Execute   :=FALSE,
	 Axis	:=Master.Axis,
);
Master.fbMC_MoveRelative[2](
	Execute   :=FALSE,
	 Axis	:=Master.Axis
);

	FOR idx:=1 TO No DO
		IF AxisIsOn[idx] THEN
			CASE EMGStopState[idx] OF
				S_DisableSetPointGenerator:
					Axis[idx].DisableSetPointGenerator(Execute := TRUE, Axis :=  Axis[idx].Axis);
					IF Axis[idx].DisableSetPointGenerator.Done THEN
						 EMGStopState[idx] := S_STOP_DECOUPLE;
					END_IF
				S_STOP_DECOUPLE:
					(*Decouple*)
					Cam[idx].CamOut(Execute := TRUE, Slave:=Axis[idx].Axis);
					IF Cam[idx].CamOut.Done THEN
						 EMGStopState[idx] := S_STOP_HALT;
					END_IF
				S_STOP_HALT:
					(*MC_HALT*)
					HaltTrig[idx](CLK:= TRUE);
					Halt[idx](
						Execute 		:= HaltTrig[idx].Q,
						Deceleration 	:= BrakeParam[idx].Deceleration,
						Jerk 		:= BrakeParam[idx].Jerk,
						BufferMode 	:= MC_Aborting,
						Axis			:= Axis[idx].Axis
					);
					IF Halt[idx].Done OR Halt[idx].Error THEN
						EMGStopState[idx] := S_STOP_RESET;
					END_IF
				S_STOP_RESET:
					(*所有軸Reset=>停止或是清除ALARM*)
					ResetTrig[idx](CLK:= TRUE);
					Axis[idx].fbMC_Reset(
						Execute:=ResetTrig[idx].Q,
						Axis:=Axis[idx].Axis
					);
					IF Axis[idx].fbMC_Reset.Done = TRUE THEN
						EMGStopState[idx] := S_STOP_RELATIVE;
					END_IF
				S_STOP_RELATIVE:
					(*恢復手動和生產的相對運動功能*)
					Axis[idx].fbMC_MoveRelative[1](
						Execute   :=FALSE,
						 Axis	:=Axis[idx].Axis,
					);
					Axis[idx].fbMC_MoveRelative[2](
						Execute   :=FALSE,
						 Axis	:=Axis[idx].Axis
					);
					(*恢復ZRT用JOG*)
					AxisValue[idx].Jog_JogForward       := FALSE;
					AxisValue[idx].Jog_JogBackwards := FALSE;

					EMGStopState[idx] :=S_STOP_IDLE;

			END_CASE
		ELSE
			(*沒開起的軸直接IDLE*)
			EMGStopState[idx] :=S_STOP_IDLE;
		END_IF
	END_FOR

	EMGStopCompleteNum := 0;
	FOR Idx:= 1 TO No DO
		IF EMGStopState[idx] = S_STOP_IDLE THEN
			EMGStopCompleteNum := EMGStopCompleteNum + 1;
		END_IF
	END_FOR
	(*全部做完*)
	IF EMGStopCompleteNum = No THEN
		Emgstoptrig := FALSE;
		FirstTime := TRUE;
	END_IF
END_IF

END_PROGRAM

// ---- POUs/FB/RelativeMOVE.TcPOU
FUNCTION_BLOCK RelativeMOVE
VAR_INPUT
	MoveAxisIdx			: INT;
	MoveDistance		: LREAL;
	MoveVelocity			: LREAL;
	MoveAcceleration		: LREAL;
	MoveDeceleration		: LREAL;
	MoveJerk			: LREAL;
END_VAR
VAR_OUTPUT
END_VAR
VAR
END_VAR


Axis[MoveAxisIdx].fbMC_MoveRelative[1](
	Execute  		:= TRUE,
	Distance		:= MoveDistance,
	Velocity  		:= MoveVelocity,
	Acceleration   := MoveAcceleration,
	Deceleration  := MoveDeceleration,
	Jerk			:= MoveJerk,
	BufferMode     := MC_BlendingHigh,
	Axis			:= Axis[MoveAxisIdx].Axis
);

Axis[MoveAxisIdx].fbMC_MoveRelative[1](
	Execute  		:= FALSE,
	Axis			:= Axis[MoveAxisIdx].Axis
);

END_FUNCTION_BLOCK

// ---- POUs/FB/RelativeMOVE2.TcPOU
FUNCTION_BLOCK RelativeMOVE2
VAR_INPUT
	MoveAxisIdx			: INT;
	MoveDistance		: LREAL;
	MoveVelocity			: LREAL;
	MoveAcceleration		: LREAL;
	MoveDeceleration		: LREAL;
	MoveJerk			: LREAL;
END_VAR
VAR_OUTPUT
END_VAR
VAR
END_VAR


Axis[MoveAxisIdx].fbMC_MoveRelative[2](
	Execute  		:= TRUE,
	Distance		:= MoveDistance,
	Velocity  		:= MoveVelocity,
	Acceleration   := MoveAcceleration,
	Deceleration  := MoveDeceleration,
	Jerk			:= MoveJerk,
	BufferMode     := MC_BlendingHigh,
	Axis			:= Axis[MoveAxisIdx].Axis
);

Axis[MoveAxisIdx].fbMC_MoveRelative[2](
	Execute  		:= FALSE,
	Axis			:= Axis[MoveAxisIdx].Axis
);

END_FUNCTION_BLOCK

// ---- POUs/FB/FB_CloseOil.TcPOU
FUNCTION_BLOCK FB_CloseOil
VAR_INPUT
END_VAR
VAR_OUTPUT
END_VAR
VAR
	idx			: INT;
END_VAR

FOR idx:=1 TO OilNo DO
	Oil[idx].IsOpen := FALSE;
	Oil[idx].CurTime := 0;
	Oil[idx].CloseStrokes := 0;
END_FOR

END_FUNCTION_BLOCK

// ---- POUs/Error.TcPOU
PROGRAM Error
VAR
	ENUMERRORSTATE :(S_ERROR_DisableSetPointGenerator, S_ERROR_DECOUPLE, S_ERROR_HALT, S_ERROR_RESET, S_ERROR_RELATIVE, S_ERROR_IDLE);
	ErrorProState		   : ARRAY [1..No] OF INT;
	idx 				   : INT:=0;
	RelativeError		   : BOOL:=FALSE;
	PowerError		   : BOOL:=FALSE;
	IOError			   : BOOL:=FALSE;
	EcSlaveError	   : BOOL:=FALSE;
	HaltTrig			   : ARRAY [1..No] OF R_TRIG;
	MasterResetTrig	   : R_TRIG;
	FeederSetTrig	   : R_TRIG;
	ResetTrig		   : ARRAY [1..No] OF R_TRIG;
	ResetTrigByUI	   : ARRAY [1..No] OF R_TRIG;
	ResetByUI		   : BOOL:=FALSE;
	ErrorTrig		  	   : R_TRIG;
	ReadAxisError	   : MC_ReadStatus;
	AxisStatusErrorID	   : ARRAY [1..No] OF DWORD;
	AxisRelativeErrorID : ARRAY [1..No] OF UDINT;
	ResetTimer		   : TON;
	CloseOil			   : FB_CloseOil;
	ToubleShootIsError : FB_ToubleShootIsError;
	IsEcAbnormal	   : FB_EcAbnormal;
END_VAR



IF ResetByUI = TRUE THEN
	BuzzerIsOpen     := FALSE;(*蜂鳴器關*)
	RelativeError      :=FALSE;
	PowerError    	    :=FALSE;
	IOError  	      	    := FALSE;
	EcSlaveError	:= FALSE;
	TouchMissStop := FALSE;
	IsConnecting	:= TRUE;
	ErrorTrig(CLK:=FALSE);

	(*F軸跳機先設位置再Reset*)
	IF AlarmList.FAlarm_1370 THEN
		FeederSetTrig(CLK:=TRUE);
		IF FeederSetTrig.Q THEN
			Axis[FeederNo].fbMC_SetPosition(
				Execute	:= FeederSetTrig.Q,
				Position	:= 0,
				Axis		:= Axis[FeederNo].Axis
			);
		END_IF
		IF Axis[FeederNo].fbMC_SetPosition.Done THEN
			FAlarmReset := TRUE;
		END_IF
	END_IF

	(*UIReset*)
MasterResetTrig(CLK:= FALSE);
	FOR idx:=1 TO No DO
		IF AxisIsOn[idx] THEN
			(*清除錯誤訊息*)
			HaltTrig[idx](CLK:=FALSE);
			ResetTrig[idx](CLK:= FALSE);
			AxisStatusErrorID[idx]	   :=0;
			AxisRelativeErrorID[idx]  :=0;
			ErrorProState[idx]		   :=S_ERROR_DisableSetPointGenerator;
			(*ResetAlarm*)
			ResetTrigByUI[idx](CLK:=TRUE);
			Axis[idx].fbMC_Reset(
				Execute:=ResetTrigByUI[idx].Q,
				Axis:=Axis[idx].Axis
			);
		END_IF
	END_FOR

	(*------AlarmList清除------*)
	AlarmListClear := TRUE;

	(*Reset延遲500ms才繼續*)
	ResetTimer(IN:= TRUE,PT:= T#500ms );
	IF ResetTimer.Q = TRUE THEN
		ResetTimer(IN:= FALSE);
		FeederSetTrig(CLK:=FALSE);

		FAlarmReset := FALSE;

		FOR idx:=1 TO No DO
			ResetTrigByUI[idx](CLK:=FALSE);
		END_FOR
		ResetByUI := FALSE;
	END_IF

ELSE

	(*檢查是否有Error*)
	IF State = ENUMSTATE.S_TROUBLESHOOT OR State = ENUMSTATE.S_TROSHO_MANMOV THEN
		RelativeError := FALSE;
		PowerError     := FALSE;
	END_IF
	FOR idx:=1 TO No DO
		IF AxisIsOn[idx] THEN
			IF ( ProAndManRelative[idx].Error[1] = TRUE ) OR ( ProAndManRelative[idx].Error[2] = TRUE ) THEN
				RelativeError:=TRUE;
			ELSIF   ( Axis[idx].fbMC_Power.Error = TRUE ) THEN
				PowerError := TRUE;
			END_IF
			IF DriveAlarmCode[idx].Error1 <> 0 OR  DriveAlarmCode[idx].Error2 <> 0 OR  DriveAlarmCode[idx].Error3 <> 0 OR  DriveAlarmCode[idx].Error4 <> 0 THEN
				PowerError := TRUE;
			END_IF
		END_IF
	END_FOR

	(*判斷是否為IO錯誤*)
	IF State = ENUMSTATE.S_TROUBLESHOOT OR State = ENUMSTATE.S_TROSHO_MANMOV THEN
		ToubleShootIsError(IsError => IOError);

		FOR idx := 0 TO MaxSlaves DO
			SlaveEcData[idx].InfoData := SlaveEcInfoData[idx];
		END_FOR
	ELSE
		IF AlarmList.Reset OR AlarmList.ExFeederError OR AlarmList.SafetyError OR  AlarmList.OilError OR AlarmList.EMGStop OR AlarmList.FAlarm_1370 OR AlarmList.ExDeviceError
		OR AlarmList.PanelEStop OR AlarmList.FrontEStop OR AlarmList.SideEStop OR AlarmList.RearEStop OR AlarmList.DecoilorEStop
		OR AlarmList.SafetyError1 OR AlarmList.SafetyError2 OR AlarmList.SafetyError3 OR AlarmList.SafetyError4 OR IsConnecting = FALSE
		OR AlarmList.NG
		THEN
			IOError := TRUE;
		END_IF
	END_IF

	IsEcAbnormal( Abnormal => EcSlaveError );

	FOR idx := 0 TO MaxSlaves DO
		SlaveEcData[idx].InfoData := SlaveEcInfoData[idx];
	END_FOR

	IF RelativeError OR PowerError OR IOError OR EcSlaveError THEN
		ErrorTrig(CLK :=TRUE);
		IF ErrorTrig.Q = TRUE THEN
			State 		:= ENUMSTATE.S_ERROR;
			(*---------- 生產部分---------*)
			Producing  	:= FALSE;(*停止生產*)
			CycleLastCmdIsRun := TRUE;
			(*--------------------------------*)
			ProFirstTime  := TRUE;
			ZRTFirstTime := TRUE;
			SubRunAloneFirstTime := TRUE;
			SubRunning	:= FALSE;
			MoveToPosFirstTime	:= TRUE;
			MoveToColPosRunning := FALSE;
						CloseOil();(*關閉油機*)
			SpeedDownTo0 := FALSE;
(*Master Reset*)
MasterResetTrig(CLK:= TRUE);
Master.fbMC_Reset(
	Execute:=MasterResetTrig.Q,
	Axis:=Master.Axis
);
Master.fbMC_MoveRelative[1](
	Execute   :=FALSE,
	 Axis	:=Master.Axis,
);
Master.fbMC_MoveRelative[2](
	Execute   :=FALSE,
	 Axis	:=Master.Axis
);
			FOR idx:=1 TO No DO
				IF AxisIsOn[idx] THEN
					(*讀取AxisError訊息*)
					(*ReadAxisError(
						Enable	 	:= TRUE,
						Axis			:= Axis[idx].Axis,
						ErrorID 		=>AxisStatusErrorID[idx]
					);*)
					 AxisStatusErrorID[idx] := Axis[idx].fbMC_Power.ErrorID;
					(*只記一組相對移動FB的錯誤*)
					AxisRelativeErrorID[idx] := Axis[idx].fbMC_MoveRelative[1].ErrorID;
					IF AxisRelativeErrorID[idx]=0 THEN
						AxisRelativeErrorID[idx] := Axis[idx].fbMC_MoveRelative[2].ErrorID;
					END_IF
				END_IF
			END_FOR

		END_IF

		FOR idx:=1 TO No DO
			IF AxisIsOn[idx] THEN
				CASE ErrorProState[idx] OF
					S_ERROR_DisableSetPointGenerator:
						Axis[idx].DisableSetPointGenerator(Execute := TRUE, Axis :=  Axis[idx].Axis);
						IF Axis[idx].DisableSetPointGenerator.Done THEN
							 ErrorProState[idx] := S_ERROR_DECOUPLE;
						END_IF
					S_ERROR_DECOUPLE:
						(*Decouple*)
						Cam[idx].CamOut(Execute := TRUE, Slave:=Axis[idx].Axis);
						IF Cam[idx].CamOut.Done THEN
							 ErrorProState[idx] := S_ERROR_HALT;
						END_IF
					S_ERROR_HALT:
						(*MC_HALT*)
						HaltTrig[idx](CLK:= TRUE);
						Halt[idx](
							Execute 		:= HaltTrig[idx].Q,
							Deceleration 	:= BrakeParam[idx].Deceleration,
							Jerk 		:= BrakeParam[idx].Jerk,
							BufferMode 	:= MC_Aborting,
							Axis			:= Axis[idx].Axis
						);
						IF Halt[idx].Done OR Halt[idx].Error THEN
							(*ErrorProState[idx] := S_ERROR_RESET;*)
							ErrorProState[idx] := S_ERROR_RELATIVE;
						END_IF
(*					S_ERROR_RESET:
						(*所有軸Reset=>停止或是清除ALARM*)
						ResetTrig[idx](CLK:= TRUE);
						Axis[idx].fbMC_Reset(
							Execute:=ResetTrig[idx].Q,
							Axis:=Axis[idx].Axis
						);
						IF Axis[idx].fbMC_Reset.Done = TRUE THEN
							ErrorProState[idx] := S_ERROR_RELATIVE;
						END_IF
*)
					S_ERROR_RELATIVE:
						(*恢復手動和生產的相對運動功能*)
						Axis[idx].fbMC_MoveRelative[1](
							Execute   :=FALSE,
							 Axis	:=Axis[idx].Axis,
						);
						Axis[idx].fbMC_MoveRelative[2](
							Execute   :=FALSE,
							 Axis	:=Axis[idx].Axis
						);
						(*恢復ZRT用JOG*)
						AxisValue[idx].Jog_JogForward       := FALSE;
						AxisValue[idx].Jog_JogBackwards := FALSE;

						ErrorProState[idx] :=S_ERROR_IDLE;

				END_CASE
			END_IF
		END_FOR

	ELSE

		IF State = ENUMSTATE.S_ERROR OR State = ENUMSTATE.S_TROUBLESHOOT THEN

			BuzzerIsOpen       := FALSE;(*蜂鳴器關*)
			RelativeError      := FALSE;
			PowerError    	   := FALSE;
			IOError  	       := FALSE;
			TouchMissStop      := FALSE;
			IsUseVROverride    := FALSE;
			IsVirtualOOverride := FALSE;
			ErrorTrig(CLK:=FALSE);(* PLC沒改到 *)
			(*UIReset*)
			MasterResetTrig(CLK:= FALSE);
			FOR idx:=1 TO No DO
				IF AxisIsOn[idx] THEN
					(*清除錯誤訊息*)
					HaltTrig[idx](CLK:=FALSE);
					ResetTrig[idx](CLK:= FALSE);
					AxisStatusErrorID[idx]	   :=0;
					AxisRelativeErrorID[idx]  :=0;
					ErrorProState[idx]		   :=S_ERROR_DisableSetPointGenerator;
					(*ResetAlarm*)
					ResetTrigByUI[idx](CLK:=TRUE);
					Axis[idx].fbMC_Reset(
						Execute:=ResetTrigByUI[idx].Q,
						Axis:=Axis[idx].Axis
					);
				END_IF
			END_FOR
	
			(*------AlarmList清除------*)			
			AlarmListClear := TRUE;

			State := ENUMSTATE.S_IDLE;
		ELSIF State = ENUMSTATE.S_TROSHO_MANMOV THEN

			BuzzerIsOpen       := FALSE;(*蜂鳴器關*)
			RelativeError      := FALSE;
			PowerError    	   := FALSE;
			IOError  	       := FALSE;
			TouchMissStop 	   := FALSE;
			IsUseVROverride    := FALSE;
			IsVirtualOOverride := FALSE;
			ErrorTrig(CLK:=FALSE);(* PLC沒改到 *)
			(*UIReset*)
			MasterResetTrig(CLK:= FALSE);
			FOR idx:=1 TO No DO
				IF AxisIsOn[idx] THEN
					(*清除錯誤訊息*)
					HaltTrig[idx](CLK:=FALSE);
					ResetTrig[idx](CLK:= FALSE);
					AxisStatusErrorID[idx]	   :=0;
					AxisRelativeErrorID[idx]  :=0;
					ErrorProState[idx]		   :=S_ERROR_DisableSetPointGenerator;
					(*ResetAlarm*)
					ResetTrigByUI[idx](CLK:=TRUE);
					Axis[idx].fbMC_Reset(
						Execute:=ResetTrigByUI[idx].Q,
						Axis:=Axis[idx].Axis
					);
				END_IF
			END_FOR
	
			(*------AlarmList清除------*)			
			AlarmListClear := TRUE;

			State := ENUMSTATE.S_MANMOV;
		END_IF
	END_IF

END_IF

END_PROGRAM

// ---- POUs/FB/FB_ToubleShootIsError.TcPOU
FUNCTION_BLOCK FB_ToubleShootIsError
VAR_INPUT
END_VAR
VAR_OUTPUT
	IsError	: BOOL;
END_VAR
VAR
END_VAR

IsError := FALSE;
IF Inputstate.Reset OR Inputstate.ExFeederError  OR  Inputstate.OilError OR Inputstate.EMGStop OR Inputstate.FAlarm_1370 OR Inputstate.ExDeviceError
OR Inputstate.PanelEStop OR Inputstate.FrontEStop OR Inputstate.SideEStop OR Inputstate.RearEStop OR Inputstate.DecoilorEStop OR IsConnecting = FALSE
OR Inputstate.NG
THEN
	IsError := TRUE;
END_IF
IF IOSwitch.SaftyEnable 
AND (Inputstate.SafetyError OR Inputstate.SafetyError1 OR Inputstate.SafetyError2 OR Inputstate.SafetyError3 OR Inputstate.SafetyError4)
THEN
	IsError := TRUE;
END_IF

END_FUNCTION_BLOCK

// ---- POUs/FB/FB_EcAbnormal.TcPOU
FUNCTION_BLOCK FB_EcAbnormal
VAR_INPUT

END_VAR
VAR_OUTPUT
	Abnormal	   :BOOL;
END_VAR
VAR
    idx            :INT;
    paxis          :INT;
    useCU1128      :BOOL;
    DriveInfoData  :ARRAY [1..No] OF UINT;
END_VAR


paxis    := 1;
Abnormal := FALSE;
useCU1128:= FALSE;
FOR idx:=0 TO MaxSlaves DO

    IF SlaveConfigData[idx].sType = 'CU1128' THEN
        useCU1128 := TRUE;
    END_IF

    IF SlaveConfigData[idx].sType = 'SanyoDenki RS2 ' OR SlaveConfigData[idx].sType = 'SGD7S-xxxxA0x C' THEN

        IF paxis <= No THEN
            DriveInfoData[paxis] := SlaveEcInfoData[idx];
            IF DriveInfoData[paxis] > 8 THEN
                IF (MachineType = MachineTypeEnum._1020 AND paxis > 10) OR paxis > 11 THEN (* 表示已經是CU1128/標準11軸 後面的軸都當作是Extension軸 *)
                    IF AxisIsOn[paxis] THEN
                        IF ((UINT_TO_WORD(DriveInfoData[paxis]) AND 16#2200) = 16#2200) OR
                        ((UINT_TO_WORD(DriveInfoData[paxis]) AND 16#2400) = 16#2400)
                        THEN
                            ;
                        ELSE
                            Abnormal := TRUE;
                        END_IF
                    END_IF
                ELSE
                    Abnormal := TRUE;
                END_IF
            END_IF            
        END_IF
        paxis := paxis + 1;

    ELSE
        IF SlaveEcInfoData[idx] > 8
        AND SlaveConfigData[idx].sType <> 'CU1128'
		AND SlaveConfigData[idx].sType <> 'CU1128-B'
		AND SlaveConfigData[idx].sType <> 'CU1128-C'
		THEN
            Abnormal := TRUE;
        END_IF

    END_IF

END_FOR

END_FUNCTION_BLOCK

// ---- POUs/FB/AlarmListClear.TcPOU
FUNCTION_BLOCK AlarmListClear
VAR_INPUT
END_VAR
VAR_OUTPUT
END_VAR
VAR
END_VAR


AlarmList.Reset := FALSE;
AlarmList.OilError := FALSE;
AlarmList.ExFeederError := FALSE;
AlarmList.SafetyError := FALSE;
AlarmList.EMGStop := FALSE;
AlarmList.FAlarm_1370 := FALSE;
AlarmList.ExDeviceError := FALSE;

END_FUNCTION_BLOCK

// ---- POUs/prAxis.TcPOU
PROGRAM prAxis
VAR
	idx				: INT ;
	RCount1			: UINT:=0;
	RCount2			: UINT:=0;
END_VAR

aprPowerST();
aprRelativeST();
aprRelativeST2();
aprReadStatusST();
aprSetPositionST();
aprJogST();
aprReadActualPosition();
aprTouchProbe();
aprCamIn();
aprCamOut();
aprCamTableSelect();
aprExtSetPointGenerator();

ACTION aprCamIn:
FOR idx :=1 TO No DO
	Cam[idx].Scaling.MasterScaling := 1000.0;
	(*Cam[idx].Scaling.MasterRelative := FALSE;*)
	Cam[idx].Scaling.MasterScalingMode := MC_CAMSCALING_AUTOOFFSET;
	Cam[idx].Scaling.SlaveScaling   := 1;
	(*Cam[idx].Scaling.SlaveRelative   := TRUE;*)
	Cam[idx].Scaling.SlaveScalingMode := MC_CAMSCALING_AUTOOFFSET;
	Cam[idx].Options.InterpolationType := MC_INTERPOLATIONTYPE_LINEAR;
	Cam[idx].Options.CamOperationMode := CAMOPERATIONMODE_EXCHANGE;

	Cam[idx].CamIn(
		Scaling			:= Cam[idx].Scaling,
		Options			:= Cam[idx].Options,
		Master		 	:= Master.Axis,
		Slave		 	:= Axis[idx].Axis,
	);
END_FOR;
END_ACTION

ACTION aprCamOut:
FOR idx := 1 TO No DO
	Cam[idx].CamOut(Slave :=  Axis[idx].Axis);

	IF Cam[idx].CamOut.Done = TRUE THEN
		Cam[idx].CamOut.Execute := FALSE;
	END_IF
END_FOR
END_ACTION

ACTION aprCamTableSelect:
FOR idx :=1 TO No DO

	Cam[idx].TableSelect(
		CamTableID     := idx,
		Master		   := Master.Axis,
		Slave		   := Axis[idx].Axis,
		CamTable	   := Cam[idx].Table
	);

	Cam[idx].TableSelect2(
		CamTableID     := idx+No,
		Master		   := Master.Axis,
		Slave		   := Axis[idx].Axis,
		CamTable	   := Cam[idx].Table2
	);

END_FOR;
END_ACTION

ACTION aprExtSetPointGenerator:
FOR idx := 1 TO No DO
	(*Enable*)
	Axis[idx].EnableSetPointGenerator(Axis :=  Axis[idx].Axis);
(*	IF Axis[idx].EnableSetPointGenerator.Done = TRUE THEN
		Axis[idx].EnableSetPointGenerator.Execute := FALSE;
	END_IF
*)
	(*Disable*)
	Axis[idx].DisableSetPointGenerator(Axis :=  Axis[idx].Axis);
	IF Axis[idx].DisableSetPointGenerator.Done THEN
		Axis[idx].DisableSetPointGenerator.Execute := FALSE;
	END_IF

END_FOR
END_ACTION

ACTION aprJogST:
FOR idx :=1 TO No DO

	Axis[idx].fbMC_Jog(
		JogForward		:= AxisValue[idx].Jog_JogForward,
		JogBackwards	:= AxisValue[idx].Jog_JogBackwards,
		Mode 			:= AxisValue[idx].Jog_Mode,
		Position 			:= AxisValue[idx].Jog_Position,
		Velocity 			:= AxisValue[idx].Jog_Velocity,
		Acceleration 		:= AxisValue[idx].Jog_Acceleration,
		Deceleration		:= AxisValue[idx].Jog_Deceleration,
		Jerk 			:= AxisValue[idx].Jog_Jerk,
		Axis				:= Axis[idx].Axis
	);

END_FOR;
END_ACTION

ACTION aprPowerST:
Master.fbMC_Power(
		Enable			:=TRUE,
		Enable_Negative 	:=TRUE,
		Enable_Positive	:=TRUE,
		Override 			:= 100,
		Axis				:=Master.Axis
);

FOR idx :=1 TO No DO
	Axis[idx].fbMC_Power(
		Enable			:=TRUE,
		Enable_Negative 	:=TRUE,
		Enable_Positive	:=TRUE,
		Override 			:= 100,
		Axis				:=Axis[idx].Axis
	);
	Axis[idx].stPowerMcOutputs.Done		:=Axis[idx].fbMC_Power.Status;
	Axis[idx].stPowerMcOutputs.Busy		:=Axis[idx].fbMC_Power.Busy;
	Axis[idx].stPowerMcOutputs.Active   		:=Axis[idx].fbMC_Power.Active;
	Axis[idx].stPowerMcOutputs.Error  		:=Axis[idx].fbMC_Power.Error;
	Axis[idx].stPowerMcOutputs.ErrorID		:=Axis[idx].fbMC_Power.ErrorID;

END_FOR;
END_ACTION

ACTION aprReadActualPosition:
Master.fb_MC_ReadActualPosition(
		Enable 		:= TRUE,
		Axis			:= Master.Axis,
		Position		=>Master.ActPos
);

FOR idx :=1 TO No DO

	Axis[idx].fb_MC_ReadActualPosition(
		Enable 		:= TRUE,
		Axis			:= Axis[idx].Axis,
		Position		=>Axis[idx].ActPos
	);

END_FOR;
END_ACTION

ACTION aprReadStatusST:
FOR idx:=1 TO No DO
	Axis[idx].fbMC_ReadStatus(
		Enable := TRUE,
		Axis       := Axis[idx].Axis
	);
END_FOR
END_ACTION

ACTION aprRelativeST:
Master.fbMC_MoveRelative[1](
	Axis	:= Master.Axis,
);

FOR idx :=1 TO No DO
	Axis[idx].fbMC_MoveRelative[1](
		Axis					:= Axis[idx].Axis,

		Done				=> ProAndManRelative[idx].Done[1],
		Busy				=> ProAndManRelative[idx].Busy[1],
		Active				=> ProAndManRelative[idx].Active[1],
		CommandAborted		=> ProAndManRelative[idx].CommandAborted[1],
		Error				=> ProAndManRelative[idx].Error[1],
		ErrorID				=> ProAndManRelative[idx].ErrorID[1]
	);
	(*IF Axis[idx].fbMC_MoveRelative[1].Done = TRUE THEN
		Axis[idx].fbMC_MoveRelative[1].Execute :=FALSE;
	END_IF;*)
END_FOR;
END_ACTION

ACTION aprRelativeST2:
Master.fbMC_MoveRelative[2](
	Axis	:= Master.Axis,
);

FOR idx :=1 TO No DO
	Axis[idx].fbMC_MoveRelative[2](
		Axis			:= Axis[idx].Axis,

		Done				=> ProAndManRelative[idx].Done[2],
		Busy				=> ProAndManRelative[idx].Busy[2],
		Active				=> ProAndManRelative[idx].Active[2],
		CommandAborted		=> ProAndManRelative[idx].CommandAborted[2],
		Error				=> ProAndManRelative[idx].Error[2],
		ErrorID				=> ProAndManRelative[idx].ErrorID[2]
	);
	(*IF Axis[idx].fbMC_MoveRelative[2].Done = TRUE THEN
		Axis[idx].fbMC_MoveRelative[2].Execute :=FALSE;
	END_IF;*)
END_FOR;
END_ACTION

ACTION aprSetPositionST:
Master.fbMC_SetPosition(Axis:=Master.Axis);
IF Master.fbMC_SetPosition.Done = TRUE THEN
	Master.fbMC_SetPosition.Execute := FALSE;
END_IF

FOR idx := 1 TO No DO
	Axis[idx].fbMC_SetPosition(Axis:=Axis[idx].Axis);

	IF Axis[idx].fbMC_SetPosition.Done = TRUE THEN
		Axis[idx].fbMC_SetPosition.Execute := FALSE;
	END_IF
END_FOR
END_ACTION

ACTION aprTouchProbe:
FOR idx:=1 TO No DO
	AxisTouchProbe[idx].Trigger_Ref.EncoderID		 := idx;
	AxisTouchProbe[idx].Trigger_Ref.TouchProbe		 := PlcEvent;
	//AxisTouchProbe[idx].Trigger_Ref.PlcEvent		 := DigInSlave[1].Input[idx-1];
	AxisTouchProbe[idx].Trigger_Ref.SignalSource	 := SignalSource_ZeroPulse;
	AxisTouchProbe[idx].Trigger_Ref.Mode			 := TOUCHPROBEMODE_SINGLE;
	Axis[idx].fbMC_TouchProbe(
		Execute	      	         	         := AxisTouchProbe[idx].Execute,
		WindowOnly			:= AxisTouchProbe[idx].WindowOnly,
		FirstPosition			:= AxisTouchProbe[idx].FirstPosition,
		LastPosition		 	:= AxisTouchProbe[idx].LastPosition,
		Axis					:= Axis[idx].Axis,
		TriggerInput   		         := AxisTouchProbe[idx].Trigger_Ref,

		RecordedPosition	         => AxisTouchProbe[idx].RecordPosition
	);
	IF AxisTouchProbe[idx].Execute=TRUE THEN
		AxisTouchProbe[idx].Execute := FALSE;
	END_IF
END_FOR;
END_ACTION

END_PROGRAM

// ---- POUs/CommunicationQualityCheck.TcPOU
PROGRAM CommunicationQualityCheck
VAR
	ClearError							: BOOL;
	IsError								: BOOL;
	LostFrames							: UDINT;
	DevState							: WORD;

	EcGetMasterDevState					: FB_EcGetMasterDevState;
	EcMasterFrameStatistic				: FB_EcMasterFrameStatistic;
	EcGetAllSlaveCrcErrors				: FB_EcGetAllSlaveCrcErrors;
	EcGetSlaveCrcErrorEx					: ARRAY[0..MaxSlaves] OF FB_EcGetSlaveCrcErrorEx;

	lastCrcErrorBuf						: ARRAY[0..MaxSlaves] OF DWORD;
	crcErrorBuf					      		: ARRAY[0..MaxSlaves] OF DWORD;
	portError								: ARRAY[0..MaxSlaves] OF ST_EcCrcErrorEx;

	firstTime								: BOOL := TRUE;
	idx									: INT;
	counter500ms							: INT:=0;
	execute								: BOOL := TRUE;
	masterDevStateString					: STRING;
	lastlostFrames						: UDINT;
END_VAR


IF counter500ms = 500 THEN
	counter500ms := 0;
	execute := FALSE;
ELSE
	execute := TRUE;
END_IF
counter500ms := counter500ms + 1;

IF ClearError THEN
	ClearError := FALSE;
	IsError 	   := FALSE;
	devState    := 0;
	firstTime     := TRUE;
END_IF

EcGetMasterDevState(
	sNetId:= DeviceNetId,
	bExecute:= execute,
	tTimeout:= ,
	bBusy=> ,
	bError=> ,
	nErrId=> ,
	nDevState=> );
IF EcGetMasterDevState.nDevState <> 0 THEN
	IsError := TRUE;
	devState := EcGetMasterDevState.nDevState;
END_IF

EcMasterFrameStatistic(
	sNetId:= DeviceNetId,
	bExecute:= execute,
	tTimeout:= ,
	bBusy=> ,
	bError=> ,
	nErrId=> ,
	nLostFrames=> lostFrames,
	fFramesPerSecond=> ,
	nLostQueuedFrames=> ,
	fQueuedFramesPerSecond=> );
IF lastLostFrames <> lostFrames AND lostFrames <> 0 THEN
	IsError := TRUE;
	lastLostFrames := lostFrames;
END_IF

EcGetAllSlaveCrcErrors(
	sNetId:= DeviceNetId,
	pCrcErrorBuf:= ADR(crcErrorBuf),
	cbBufLen:= SIZEOF(crcErrorBuf[0])* (MaxSlaves + 1),
	bExecute:= execute,
	tTimeout:= ,
	bBusy=> ,
	bError=> ,
	nErrId=> ,
	nSlaves=> );
IF firstTime THEN
	firstTime := FALSE;
	FOR idx := 0 TO MaxSlaves DO
		lastCrcErrorBuf[idx] := crcErrorBuf[idx];
	END_FOR
ELSE
	FOR idx := 0 TO MaxSlaves DO
		IF lastCrcErrorBuf[idx] <> crcErrorBuf[idx] AND crcErrorBuf[idx] <> 0 THEN
			IsError := TRUE;
			lastCrcErrorBuf[idx] := crcErrorBuf[idx];
			EcGetSlaveCrcErrorEx[idx](
				sNetId:= DeviceNetId,
				nSlaveAddr:= SlaveConfigData[idx].nAddr,
				bExecute:= TRUE,
				tTimeout:= ,
				bBusy=> ,
				bError=> ,
				nErrId=> ,
				crcError=> portError[idx]);
		ELSE
			EcGetSlaveCrcErrorEx[idx](bExecute:= FALSE, crcError=> portError[idx]);
			SlaveEcData[idx].PortA := portError[idx].portA;
			SlaveEcData[idx].PortB := portError[idx].portB;
			SlaveEcData[idx].PortC := portError[idx].portC;
			SlaveEcData[idx].PortD := portError[idx].portD;
		END_IF
	END_FOR
END_IF

END_PROGRAM

// ---- POUs/SetCountPosToActPos.TcPOU
PROGRAM SetCountPosToActPos
VAR
	idx 				: INT;
	Trig				: ARRAY [1..No] OF R_TRIG;
	SetComplete		: ARRAY [1..No] OF BOOL:=[No(FALSE)];
	SetCount			: INT:=0;
	CompleteCount	: INT:=0;
END_VAR


FOR idx:=1 TO No DO

	IF SetAxisPosByCountPos[idx] THEN
		Trig[idx](CLK:=TRUE);
		Axis[idx].fbMC_SetPosition(
			Execute	:= Trig[idx].Q,
			Position	:= AxisCountPosByInput[idx],
			Axis		:= Axis[idx].Axis
		);

		IF Axis[idx].fbMC_SetPosition.Done THEN
			SetComplete[idx] := TRUE;
		END_IF
	END_IF

END_FOR

SetCount		    := 0;
CompleteCount := 0;

FOR idx:=1 TO No DO
	IF SetAxisPosByCountPos[idx] THEN
		SetCount := SetCount + 1;
	END_IF
	IF SetComplete[idx] THEN
		CompleteCount := CompleteCount + 1;
	END_IF
END_FOR

IF CompleteCount = SetCount AND SetCount<>0 THEN
	FOR idx:=1 TO No DO
		SetAxisPosByCountPos[idx] := FALSE;
		SetComplete[idx] := FALSE;
		Trig[idx](CLK:=FALSE);
	END_FOR
	UISetPosAllComplete := TRUE;
END_IF

END_PROGRAM

// ---- POUs/Mpg.TcPOU
PROGRAM Mpg
VAR
	Value			: UINT;
	Count			: INT:=0;
	Count50MS		: INT:=0;
	CountP 			: INT:=0;
	CountN 			: INT:=0;
	CountStop		: INT:=0;
END_VAR

IF Count = 0 THEN
	Count := 1;
	Value :=  EL5101SlaveValue;
END_IF

Count50MS := Count50MS + 1;

IF Count50MS = 5 THEN
	Count50MS := 0;
	IF UINT_TO_INT( EL5101SlaveValue - Value) > 3 THEN
		CountP := CountP + 1;
		Value := EL5101SlaveValue;
		Mpg_NegativeMove := FALSE;
		Mpg_PositiveMove := TRUE;
	ELSIF UINT_TO_INT( EL5101SlaveValue - Value) < -3 THEN
		CountN := CountN + 1;
		Value :=  EL5101SlaveValue;
		Mpg_PositiveMove := FALSE;
		Mpg_NegativeMove := TRUE;
	ELSE
		CountStop := CountStop + 1;
		Mpg_PositiveMove   := FALSE;
		Mpg_NegativeMove := FALSE;
	END_IF
END_IF

END_PROGRAM

// ---- POUs/SetOverride.TcPOU
PROGRAM SetOverride
VAR
	ProduceSpeed	: INT:= 0;
	VRSpeed 		: REAL;
	TestSpeed		: INT:=0;
	MPGRate			: LREAL :=0;
	idx				: INT;
END_VAR

VRSpeed := EL3062_VR/26350.0;
IF VRSpeed < 0.01 THEN
	VRSpeed := 0;
ELSIF VRSpeed > 1 THEN
	VRSpeed := 1;
END_IF

IF State = ENUMSTATE.S_AUTO THEN
	Override := ProduceSpeed;

ELSIF State = ENUMSTATE.S_TEST THEN
	TestSpeed := LREAL_TO_INT(ProduceSpeed * VRSpeed);

	IF MachineSubType = MachineSubTypeEnum.CE AND IOSwitch.SaftyEnable (*CE要降速度 不超過30%*)
	AND (Inputstate.SafetyError1 OR Inputstate.SafetyError2 OR Inputstate.SafetyError3 OR Inputstate.SafetyError4) 
	THEN
		TestSpeed := SEL(TestSpeed > 30, TestSpeed, 30);
	END_IF

	Override := TestSpeed;

ELSIF State = ENUMSTATE.S_MPG THEN
	IF Mpg_PositiveMove = TRUE THEN
		MPGRate := SEL(MPGRate + 0.25 > 10, MPGRate + 0.25, 10);
	ELSE
		MPGRate := SEL(MPGRate - 0.25 < 0, MPGRate - 0.25, 0);
	END_IF
	Override := MPGRate;

ELSIF SubRunning THEN
	Override := LREAL_TO_INT(100 * VRSpeed);

ELSIF MoveToColPosRunning THEN
	Override := LREAL_TO_INT(20 * VRSpeed);

END_IF

IF IsVirtualOOverride THEN
	FOR idx:=1 TO NO DO
	 	Axis[idx].fbMC_SetOverride(
			Enable		:= TRUE,
			VelFactor	:= Override,
			AccFactor 	:= 1,
			JerkFactor 	:= 1,
			Axis		:= Axis[idx].Axis,
		);
	END_FOR
ELSIF IsUseVROverride THEN
	FOR idx:=1 TO NO DO
	 	Axis[idx].fbMC_SetOverride(
			Enable		:= TRUE,
			VelFactor	:= VRSpeed,
			AccFactor 	:= 1,
			JerkFactor 	:= 1,
			Axis		:= Axis[idx].Axis,
		);
	END_FOR
ELSE
	FOR idx:=1 TO NO DO
	 	Axis[idx].fbMC_SetOverride(
			Enable		:= TRUE,
			VelFactor	:= 1,
			AccFactor 	:= 1,
			JerkFactor 	:= 1,
			Axis		:= Axis[idx].Axis,
		);
	END_FOR
END_IF

END_PROGRAM

// ---- POUs/Produce.TcPOU
PROGRAM Produce
VAR
	ENUMPRODUCESTATE	:(S_FillAxisTable, S_FillSubTable, S_FillTouchAdjustTable, S_FillIOTable, S_FillSubIOTable,  S_EnableExtSetPoint, S_WaitExtSetPoint, S_Run);
	ProduceState		: INT;
	idx					: INT ;
	CloseIO				: FB_CloseIO;
	StartProNum			: UDINT;
	ProduceTimer		: UDINT:=0;
	ProduceNum			: UDINT:=1;
	ProduceCurNum		: UDINT:=0;
	UIStop				: BOOL:=FALSE;
	FlashModeOn		: BOOL;
	PPM				: REAL;
	PPMCal				: PPMCal;
	Speed				: LREAL;
	SpeedUPToOverride	: BOOL;
	SpeedCtrlAccTimer	: TON;
	SpeedCtrlDecTimer	: TON;
	SpeedAccDccTime 	: TIME := T#300ms;


	RepeatA				: DINT;
	RepeatB				: DINT;
	JumpFirstTime		: BOOL;
	StopTiming1			: DINT;
	StopTiming2			: DINT;
	JumpTiming			: DINT;
	TotalTimeByMs		: LREAL;
	CurrentTableIdx		: DINT;
	CurrentTableOffset	: REAL;
	LastTableOffset		: REAL;
	RepeatA_FeederIdx	: INT;
	Idx0FirstTime			: BOOL;

	axisIdx				: INT;
	touchIdx			: INT;
	airIdx				: INT;
	SendOffset			: UDINT := 0;
	touchTableFill 		: BOOL := FALSE;
	airTableFill  		: BOOL := FALSE;
	exFSpdUpTableFill	: BOOL := FALSE;
	receiveAllBuf		: BOOL := FALSE;
	TouchBeforeStart	: BOOL:= FALSE;
	getSubNo			: INT;

	IsExtSetPointDone	: ARRAY [1..No] OF BOOL;
	IsSetPointComplete 	: BOOL;
	TableOffsetPos		: ARRAY [1..No] OF  LREAL;
	OldPosition			: ARRAY [1..No] OF LREAL;
	ExtVelocity			: ARRAY [1..No] OF LREAL;
	OldVelocity			: ARRAY [1..No] OF LREAL;
	ExtAcceleration		: LREAL;
	ExtDirection		: DINT;
	newPos				: LREAL;

	ModuloBase			: ARRAY [1..No] OF LREAL;

	Feeder				: ST_FeederInProduce;
	FeederStartIdx		: ARRAY [0..999] OF DINT;
	FeederEndIdx		: ARRAY [0..999] OF DINT;
	FeederIdx			: INT := 0;
	FTouchShowPos		: LREAL;
	TouchDist			: ARRAY [1.. TouchNo] OF LREAL;
	IsTouch				: BOOL;
	TouchOpenNo		: UINT;
	TouchMissNum		: UDINT := 0;
	TouchMissSetNum		: UDINT := 0;
	TouchMiss			: BOOL := FALSE;
	TouchConfig			: ARRAY [1..TouchNo] OF ST_TouchConfig;
	TouchConfigIdx		: ARRAY [1..TouchNo] OF  INT;
	RepeatA_TouchConfigIdx  : ARRAY [1..TouchNo] OF  INT;
	ThisTurnTouchMiss	: BOOL;
	ThisTurnTouchMissShow   : ARRAY [1..TouchNo] OF BOOL;
	FNeedHoldPos		: FB_FNeedHoldPos;
	TouchEnd			: FB_TouchEnd;
	InAnotherTouch		: FB_InAnotherTouch;
	IsPreTouch			: BOOL;
	PreTouchShow        : ARRAY [1..TouchNo] OF BOOL;
	GlobalTouchShow     : ARRAY [1..TouchNo] OF BOOL;
	IsOverUpBound		: BOOL;
	IsBelowDownBound	: BOOL;

	IsAdjustAxis		: FB_IsAdjustAxis;
	IsAdjustTouch		: FB_IsAdjustTouch;
	TouchAdjustIdx	    : INT;
	AdjustCounter		: ARRAY [1..TouchAdjustNo] OF REAL;
	AdjustCounterBuf	: ARRAY [1..TouchAdjustNo] OF REAL;
	AdjustPos           : LREAL;
	AdjustNextPos       : LREAL;

	RunSubProgram		: BOOL;
	RunSubNo			: INT;
	SubInFirstTime		: BOOL;
	SubTableIdx			: DINT;
	SubTableOffset		: REAL;
	FInSubStartPos		: LREAL;
	FInSubPos			: LREAL;

	G5Config				: ARRAY [1..G5ConfigNo] OF ST_G5Config;
	G5Status				: ST_G5Status;

	OilStrokeCount : ARRAY[1..OilNo] OF UDINT; (*新增 判斷圈數*)

	FirstAutoRun 			: BOOL;
	CloseOil				: FB_CloseOil;

	lState				:INT;
	SpeedChanged		:BOOL;

	IsHaveHook			: BOOL := FALSE;
	HookAxisNo			: INT := -1;
	IsHookMovable		: BOOL;

	IsTouchWithF		: BOOL;

	mem			: ARRAY [0..5000] OF LREAL;
END_VAR


(*到達生產量*)
IF  ( (ProduceCurNum=ProduceNum AND ProduceNum<>0) OR (ProduceCurNum=ProduceNum AND CurrentTableIdx = TotalTimeByMs AND TouchMissNum >= TouchMissSetNum AND TouchMissSetNum = 1 ) )
     AND Producing THEN
	FOR axisIdx:=1 TO No DO
		Axis[axisIdx].DisableSetPointGenerator.Execute := TRUE;
	END_FOR
	State				   := ENUMSTATE.S_IDLE;(*狀態改回閒置*)
		CloseIO(); (*關I/O*)
	UIStop				   := FALSE;
	Producing	       		   := FALSE;
	ProFirstTime			   := TRUE;
END_IF

(*停機按鈕*)
IF Producing AND Inputstate.StopCycle THEN
	 UIStop := TRUE;
END_IF
IF NOT Producing THEN
	UIStop := FALSE;
END_IF
IF UIStop THEN
	ProduceNum := ProduceCurNum + 1;
END_IF

(*開始生產*)
IF Producing  AND (ProduceCurNum<ProduceNum)  THEN
	(*第一次進生產*)
	IF ProFirstTime = TRUE THEN
		(*初始化*)
				Initial();
	END_IF

	CtrlSpeed();

	CASE ProduceState OF

		S_FillAxisTable:
						FillAxisTable();

		S_FillIOTable:
						FillIOTable();

		S_FillSubTable:
						FillSubTable();

		S_FillSubIOTable:
						FillSubIOTable();

		S_FillTouchAdjustTable:
						FillTouchAdjustTable();

		S_EnableExtSetPoint:
						EnableExtSetPoint();

		S_WaitExtSetPoint:
						WaitExtSetPoint();

		S_Run:

			 IF State = ENUMSTATE.S_AUTO THEN (*判斷為自動時*)
				IF FirstAutoRun = TRUE THEN
					FOR idx:=1 TO OilNo DO
						IF Oil[idx].Enable AND Oil[idx].OpenTime <> 0 THEN
							Oil[idx].IsOpen := TRUE;
						END_IF
					END_FOR
					FirstAutoRun := FALSE;
				END_IF
								OilFunc();
			ELSE
				IF FirstAutoRun = FALSE THEN
					firstAutoRun := TRUE;
										CloseOil();
				END_IF
			END_IF

			ProduceTimer := ProduceTimer + 1;

			(* 表一開始 初始*)
			IF CurrentTableIdx = 0 AND Idx0FirstTime THEN
				Idx0FirstTime 		:= FALSE;
				(*如果翻線使用虛擬原點 會造成送線表開始有一個位移要扣掉*)
				IF AxisTable1[FeederNo, 0] <> 0 THEN
					Feeder.BasePos := Feeder.CurPos - AxisTable1[FeederNo, 0];
				ELSE
					Feeder.BasePos := Feeder.CurPos;
				END_IF
				FeederIdx 		:= 0;
				Feeder.StillPos 	:= 0;
				IsTouch 			:= FALSE;
				IsPreTouch			:= FALSE;
				TouchMiss 		:= FALSE;
				ThisTurnTouchMiss := FALSE;
				TouchOpenNo 	:= 0;
				IsHookMovable		:= TRUE;
				FOR touchIdx := 1 TO TouchNo DO
					TouchDist[touchIdx]		 := 0;
					TouchConfigIdx[touchIdx] := 0;
					PreTouchShow[touchIdx]   := FALSE;
					ThisTurnTouchMissShow[touchIdx] := FALSE;
					GlobalTouchShow[touchIdx]   := FALSE;
				END_FOR
				FOR axisIdx := 1 TO No DO
					IF AxesUseModulo[axisIdx] THEN
						ModuloBase[axisIdx] :=  AxesModuloTurns[axisIdx]  *  AxesGradPerTurn[axisIdx] ;
					END_IF
				END_FOR
				FOR TouchAdjustIdx := 1 TO TouchAdjustNo DO
					AdjustCounter[TouchAdjustIdx] := AdjustCounter[TouchAdjustIdx] + AdjustCounterBuf[TouchAdjustIdx];
					AdjustCounterBuf[TouchAdjustIdx] := 0;
				END_FOR
			END_IF

			(*副程式*)
			IF RunSubNo <= SubProgramNo
			AND (SubProgramConfig[RunSubNo].Reaction = 1 OR SubProgramConfig[RunSubNo].Reaction = 2 AND ThisTurnTouchMiss)
			AND SubProgramConfig[RunSubNo].TotalTableSize <> 0
			AND CurrentTableIdx = SubProgramConfig[RunSubNo].StartIdx + 1 (*StartIdx 要+1開始 因為ThisTurnTouchMiss在StartIdx下一周期才會拿到*)
			THEN

				IF SubInFirstTime THEN
					SubInFirstTime := FALSE;
					SubTableOffset := CurrentTableOffset;
					FInSubStartPos := Feeder.CurPos;
				END_IF


				(* 設定ExtPosition *)
				FOR axisIdx := 1 TO No DO
					IF AxisIsOn[axisIdx] THEN
						(* 超過這條最後idx *)
						IF (SubTableIdx + SubTableOffset) > (SubProgramConfig[RunSubNo].TotalTableSize - 1) THEN
							TableOffsetPos[axisIdx]:= SubProgramTable[RunSubNo].AxisTable[axisIdx, SubTableIdx];
						ELSE
						(* idx在此表內 *)
							TableOffsetPos[axisIdx]:= SubProgramTable[RunSubNo].AxisTable[axisIdx, SubTableIdx] + ( SubProgramTable[RunSubNo].AxisTable[axisIdx, SubTableIdx + 1] - SubProgramTable[RunSubNo].AxisTable[axisIdx, SubTableIdx] ) * SubTableOffset;
						END_IF
					END_IF
				END_FOR

								SubAirFunc();

				FOR axisIdx := 1 TO No DO
					IF AxisIsOn[axisIdx] THEN
						(*送線處理*)
						IF axisIdx = FeederNo THEN

							FInSubPos := FInSubStartPos + TableOffsetPos[axisIdx];
							ExtVelocity[axisIdx]:= (FInSubPos - OldPosition[axisIdx]) / (UDINT_TO_LREAL(_TaskInfo[1].CycleTime) / 10000000);
							OldPosition[axisIdx]:= FInSubPos;
							ExtDirection := SEL(FInSubPos >= OldPosition[axisIdx], -1, 1);
							ExtAcceleration :=  (ExtVelocity[axisIdx] - OldVelocity[axisIdx]) / (UDINT_TO_LREAL(_TaskInfo[1].CycleTime) / 10000000);
							OldVelocity[axisIdx]:= ExtVelocity[axisIdx];

							(*Feed*)
							MC_ExtSetPointGenFeed(
								Position := FInSubPos,
								Velocity := ExtVelocity[axisIdx],
								Acceleration := ExtAcceleration,
								Direction := ExtDirection,
								Axis := Axis[axisIdx].Axis);

						(*使用Modulo軸*)
						ELSIF AxesUseModulo[axisIdx] THEN

							newPos := TableOffsetPos[axisIdx] + ModuloBase[axisIdx];

							ExtVelocity[axisIdx]:= (newPos - OldPosition[axisIdx]) / (UDINT_TO_LREAL(_TaskInfo[1].CycleTime) / 10000000);
							OldPosition[axisIdx]:= newPos;
							ExtAcceleration :=  (ExtVelocity[axisIdx] - OldVelocity[axisIdx]) / (UDINT_TO_LREAL(_TaskInfo[1].CycleTime) / 10000000);
							OldVelocity[axisIdx]:= ExtVelocity[axisIdx];
							ExtDirection := SEL(newPos >= OldPosition[axisIdx], -1, 1);

							MC_ExtSetPointGenFeed(
								Position := newPos,
								Velocity := ExtVelocity[axisIdx],
								Acceleration := ExtAcceleration,
								Direction := ExtDirection,
								Axis := Axis[axisIdx].Axis);

						(*一般軸處理*)
						ELSE
							ExtVelocity[axisIdx]:= (TableOffsetPos[axisIdx] - OldPosition[axisIdx]) / (UDINT_TO_LREAL(_TaskInfo[1].CycleTime) / 10000000);
							OldPosition[axisIdx]:= TableOffsetPos[axisIdx];
							ExtAcceleration :=  (ExtVelocity[axisIdx] - OldVelocity[axisIdx]) / (UDINT_TO_LREAL(_TaskInfo[1].CycleTime) / 10000000);
							OldVelocity[axisIdx]:= ExtVelocity[axisIdx];
							ExtDirection := SEL(TableOffsetPos[axisIdx] >= OldPosition[axisIdx], -1, 1);

							MC_ExtSetPointGenFeed(
								Position := TableOffsetPos[axisIdx],
								Velocity := ExtVelocity[axisIdx],
								Acceleration := ExtAcceleration,
								Direction := ExtDirection,
								Axis := Axis[axisIdx].Axis);
						END_IF
					END_IF
				END_FOR

				SubTableOffset := SubTableOffset + Speed/100;
				IF SubTableOffset >= 1 THEN
					SubTableOffset := SubTableOffset - 1;
					SubTableIdx := SubTableIdx + 1;
				END_IF

				IF SubTableIdx = SubProgramConfig[RunSubNo].TotalTableSize THEN
					SubTableIdx 	:= 0;
					SubInFirstTime := TRUE;
					CurrentTableOffset := SubTableOffset;

					IF SubProgramConfig[RunSubNo].Reaction = 2 THEN
						Feeder.BasePos := Feeder.BasePos + TableOffsetPos[FeederNo] + (AxisTable1[FeederNo, CurrentTableIdx] - AxisTable1[FeederNo, LREAL_TO_DINT(TotalTimeByMs - 1)]);
						CurrentTableIdx := LREAL_TO_DINT( TotalTimeByMs - 1);
					ELSE
						Feeder.BasePos := Feeder.BasePos + TableOffsetPos[FeederNo];
						IF RunSubNo <= SubProgramNo THEN
							(*重複地進入時間和副程式進入時間重疊 G5會記錄到舊的執行的副程式*)
							IF G5Config[G5Status.CurIdx].ATime + 1 = CurrentTableIdx AND G5Status.ATimeSubNo = RunSubNo THEN
								G5Status.ATimeSubNo := RunSubNo + 1;
							END_IF
							RunSubNo := RunSubNo + 1;
						END_IF						
					END_IF

				END_IF

			ELSE

			(*主程式*)
				(* 設定TableOffsetPos *)
				FOR axisIdx := 1 TO No DO
					IF AxisIsOn[axisIdx] THEN
						(* 超過這條最後idx *)
						IF (CurrentTableIdx +  CurrentTableOffset) > (TotalTimeByMs - 1) THEN
							TableOffsetPos[axisIdx]:= AxisTable1[axisIdx, CurrentTableIdx];
						ELSE
						(* idx在此表內 *)
							IsAdjustAxis(paxis := axisIdx, CurrentTableIdx := CurrentTableIdx);
							IF IsAdjustAxis.Yes THEN
								AdjustPos := AxisTable1[axisIdx, CurrentTableIdx] + TouchAdjustTable[IsAdjustAxis.AdjustIdx, CurrentTableIdx] * AdjustCounter[IsAdjustAxis.AdjustIdx];
								AdjustNextPos := AxisTable1[axisIdx, CurrentTableIdx + 1] + TouchAdjustTable[IsAdjustAxis.AdjustIdx, CurrentTableIdx + 1] * AdjustCounter[IsAdjustAxis.AdjustIdx];
								TableOffsetPos[axisIdx]:= AdjustPos + ( AdjustNextPos - AdjustPos ) * CurrentTableOffset;
							ELSE
								TableOffsetPos[axisIdx]:= AxisTable1[axisIdx, CurrentTableIdx] + ( AxisTable1[axisIdx, CurrentTableIdx + 1] - AxisTable1[axisIdx, CurrentTableIdx] ) * CurrentTableOffset;
							END_IF
						END_IF
					END_IF
				END_FOR

				(* 送線設定 *)
				IF AxisIsOn[FeederNo]THEN
					IF CurrentTableIdx = FeederStartIdx[FeederIdx] OR CurrentTableIdx = FeederEndIdx[FeederIdx] THEN
						Feeder.StillPos := AxisTable1[FeederNo, CurrentTableIdx];
					END_IF
				END_IF

								TouchFunc();
								AirFunc();
								ExFeederFunc();
				

				(* 輸入執行動作ExtSetPointGenFeed *)
				FOR axisIdx := 1 TO No DO
					IF AxisIsOn[axisIdx] THEN
						(*送線處理*)
						IF axisIdx = FeederNo THEN

							TouchEnd(CurrentIdx:=CurrentTableIdx, TouchConfig:=TouchConfig,TouchConfigIdx:=TouchConfigIdx);
							(*有探到 最後調整基準點*)
							IF TouchEnd.Yes AND (IsTouch OR IsPreTouch) THEN
								IsTouch := FALSE;
								IsPreTouch := FALSE;

								(*基準點調整, 有送線動作才調整*)
								IF IsTouchWithF THEN
									IF Feeder.TouchFeederIdx <> FeederIdx THEN
										Feeder.BasePos := Feeder.BasePos + (Feeder.TouchPos - TableOffsetPos[axisIdx]);
										Feeder.TouchPos   := AxisTable1[FeederNo, FeederEndIdx[FeederIdx]] -
															(AxisTable1[FeederNo, FeederEndIdx[Feeder.TouchFeederIdx]] - Feeder.TouchPos);
									ELSIF Feeder.TouchFeederIdx = FeederIdx THEN
										Feeder.BasePos := Feeder.BasePos + (Feeder.TouchPos - TableOffsetPos[axisIdx]);
									END_IF
								END_IF

							END_IF

														FeederPosSetting();
														FeederVelAccSetting();

							(*Feed*)
							MC_ExtSetPointGenFeed(
								Position := Feeder.CurPos,
								Velocity := ExtVelocity[axisIdx],
								Acceleration := ExtAcceleration,
								Direction := ExtDirection,
								Axis := Axis[axisIdx].Axis);
						(*夾耳軸處理*)
						ELSIF IsHaveHook AND axisIdx = HookAxisNo THEN
							
							IF IsHookMovable = FALSE THEN
								newPos := OldPosition[axisIdx];
							ELSE
								newPos := TableOffsetPos[axisIdx] + ModuloBase[axisIdx];
							END_IF
							ExtVelocity[axisIdx]:= (newPos - OldPosition[axisIdx]) / (UDINT_TO_LREAL(_TaskInfo[1].CycleTime) / 10000000);
							OldPosition[axisIdx]:= newPos;
							ExtAcceleration :=  (ExtVelocity[axisIdx] - OldVelocity[axisIdx]) / (UDINT_TO_LREAL(_TaskInfo[1].CycleTime) / 10000000);
							OldVelocity[axisIdx]:= ExtVelocity[axisIdx];
							ExtDirection := SEL(newPos >= OldPosition[axisIdx], -1, 1);

							MC_ExtSetPointGenFeed(
								Position := newPos,
								Velocity := ExtVelocity[axisIdx],
								Acceleration := ExtAcceleration,
								Direction := ExtDirection,
								Axis := Axis[axisIdx].Axis);

						(*使用Modulo軸*)
						ELSIF AxesUseModulo[axisIdx] THEN

							newPos := TableOffsetPos[axisIdx] + ModuloBase[axisIdx];

